//===================================================================//
// Ereigniskategorie - Alarmeldung - Meldung signalisiert Anlagenausfall oder erfordert sofortigen Eingriff 
// Event category - Alarm message - Message signals system failure or requires immediate intervention 
// Sicherheitstemperaturbegrenzer (STB), Sicherheitsdruckbegrenzer (SDB), Übertemperatur der Warmwasserbereitung (WWB), Sicherheitsventile, Hauptpumpen, Keilriemenwächter, Frequenzumformer, Kälteanlagen, Spannungsausfall usw
// Safety temperature limiter, safety pressure limiter, excess temperature of water heating, safety valves, main pumps, V-belt monitors, frequency converters, refrigeration systems, voltage failure, etc.
AlarmMsg.iParent							:= THIS^;
AlarmMsg.iLabel								:= LblControl_EvtCategoryAlarmMessage;									  
AlarmMsg.sObjectName						:= '{Idx=01}';
AlarmMsg.eDPADMode							:= E_BA_DPADMode.eInclude;																						
AlarmMsg.EC.nInstanceID							:= EC_ID.NC30;
AlarmMsg.EC.sObjectName							:= '{Idx=30}';
AlarmMsg.EC.eEventType							:= E_BA_EventType.eAlarm;
AlarmMsg.EC.aPriority[1]						:= 70;
AlarmMsg.EC.aPriority[2]						:= 71;
AlarmMsg.EC.aPriority[3]						:= 72;
AlarmMsg.EC.eAlarmMode						:= E_BA_AlarmMode.eExtended;	//Erweiterter Alarm


//===================================================================
// Ereigniskategorie - Störungsmeldung - Meldung weist auf einen anormalen Betriebszustand hin
// Event category - malfunction message - message indicates abnormal operating condition
// Temperaturwächter (TW), Druckwächter (DW), Temperaturüberwachung von Wärmetauscher (WT) und WWB, Motorschutz, Aufzug-Sammelstörmeldung, Netzdrücke usw.
// Temperature monitor, pressure monitor, temperature monitoring of heat exchanger and water heating, motor protection, lift collective fault signal, mains pressures, etc.
FaultMsg.iParent							:= THIS^;
FaultMsg.iLabel								:= LblControl_EvtCategoryFaultMessage;							  
FaultMsg.sObjectName						:= '{Idx=01}';
FaultMsg.eDPADMode							:= E_BA_DPADMode.eInclude;																						
FaultMsg.EC.nInstanceID							:= EC_ID.NC40;
FaultMsg.EC.sObjectName							:= '{Idx=40}';
FaultMsg.EC.eEventType							:= E_BA_EventType.eDisturb;
FaultMsg.EC.aPriority[1]						:= 100;
FaultMsg.EC.aPriority[2]						:= 101;
FaultMsg.EC.aPriority[3]						:= 102;
FaultMsg.EC.eAlarmMode						:= E_BA_AlarmMode.eStandard;	//Standard Alarm
//===================================================================
// Ereigniskategorie - Wartungsmeldung, Hinweis auf Wartungsaktivität o.ä.
// Event category - Maintenance message Maintenance message, indication of maintenance activity or similar.
// Betriebsstunden, Behälterstand, Reparaturschalter usw.
// Operating hours, tank level, repair switch, etc.
MaintenanceMsg01.iParent					:= THIS^;
MaintenanceMsg01.iLabel						:= LblControl_EvtCategoryMaintenanceMessage;									  
MaintenanceMsg01.sObjectName				:= '{Idx=01}';
MaintenanceMsg01.eDPADMode					:= E_BA_DPADMode.eInclude;																						
MaintenanceMsg01.EC.nInstanceID					:= EC_ID.NC50;
MaintenanceMsg01.EC.sObjectName					:= '{Idx=50}';
MaintenanceMsg01.EC.eEventType					:= E_BA_EventType.eMaintenance;
MaintenanceMsg01.EC.aPriority[1]				:= 130;
MaintenanceMsg01.EC.aPriority[2]				:= 131;
MaintenanceMsg01.EC.aPriority[3]				:= 132;
MaintenanceMsg01.EC.eAlarmMode						:= E_BA_AlarmMode.eStandard;	//Standard Alarm

// Filterende erreicht, Filter verschmutzt usw.
// Filter end reached, filter dirty, etc.
MaintenanceMsg02.iParent					:= THIS^;
MaintenanceMsg02.iLabel						:= LblControl_EvtCategoryMaintenanceMessage;									  
MaintenanceMsg02.sObjectName				:= '{Idx=02}';
MaintenanceMsg02.sDescription				:= '{Wartungsmeldung}';
MaintenanceMsg02.eDPADMode					:= E_BA_DPADMode.eInclude;																						
MaintenanceMsg02.EC.nInstanceID					:= EC_ID.NC51;
MaintenanceMsg02.EC.sObjectName					:= '{Idx=51}';
MaintenanceMsg02.EC.eEventType					:= E_BA_EventType.eAlarm;
MaintenanceMsg02.EC.aPriority[1]				:= 135;
MaintenanceMsg02.EC.aPriority[2]				:= 136;
MaintenanceMsg02.EC.aPriority[3]				:= 137;
MaintenanceMsg02.EC.eAlarmMode						:= E_BA_AlarmMode.eStandard;	//Standard Alarm
//===================================================================
//===================================================================
// Ereigniskategorie - Systemmeldung, Störungsmeldung aus GA-System
// Event category - System message, System message, Fault message from building automation system
// Gerätestörung, Batteriemeldung, Kommunikationsunterbrechung usw.
// Unit malfunction, battery message, communication interruption, etc.
SystemMsg.iParent							:= THIS^;
SystemMsg.iLabel							:= LblControl_EvtCategorySystem;									  
SystemMsg.sObjectName						:= '{Idx=01}';
SystemMsg.eDPADMode							:= E_BA_DPADMode.eInclude;																						
SystemMsg.EC.nInstanceID						:= EC_ID.NC60;
SystemMsg.EC.sObjectName						:= '{Idx=60}';
SystemMsg.EC.eEventType							:= E_BA_EventType.eNotification;
SystemMsg.EC.aPriority[1]						:= 180;
SystemMsg.EC.aPriority[2]						:= 181;
SystemMsg.EC.aPriority[3]						:= 182;
SystemMsg.EC.eAlarmMode						:= E_BA_AlarmMode.eSimple;	//Simple Alarm
//===================================================================//
//	Ereigniskategorie - Manual operation, Handeingriff
ManualOp.iParent							:= THIS^;
ManualOp.iLabel						 		:= LblControl_EvtCategoryManualOperation;									  
ManualOp.sObjectName						:= '{Idx=01}';
ManualOp.eDPADMode							:= E_BA_DPADMode.eInclude;																						
ManualOp.EC.nInstanceID							:= EC_ID.NC70;
ManualOp.EC.sObjectName							:= '{Idx=70}';
ManualOp.EC.eEventType							:= E_BA_EventType.eAlarm;
ManualOp.EC.aPriority[1]						:= 220;
ManualOp.EC.aPriority[2]						:= 220;
ManualOp.EC.aPriority[3]						:= 220;
ManualOp.EC.eAlarmMode						:= E_BA_AlarmMode.eSimple;	//Simple Alarm
//===================================================================//
// Ereigniskategorie - Freibleibend, Sonstige Meldungen
// Event category - Other message, Not binding, Other messages
// Betriebszustandswechsel, Betriebsarten, Trendspeicher voll usw.
// Operating status change, operating modes, trend memory full, etc.
OtherMsg.iParent							:= THIS^;
OtherMsg.iLabel						 		:= LblControl_EvtCategoryOther;									  
OtherMsg.sObjectName						:= '{Idx=01}';
OtherMsg.eDPADMode							:= E_BA_DPADMode.eInclude;																						
OtherMsg.EC.nInstanceID							:= EC_ID.NC80;
OtherMsg.EC.sObjectName							:= '{Idx=80}';
OtherMsg.EC.eEventType							:= E_BA_EventType.eAlarm;
OtherMsg.EC.aPriority[1]						:= 230;
OtherMsg.EC.aPriority[2]						:= 231;
OtherMsg.EC.aPriority[3]						:= 232;
OtherMsg.EC.eAlarmMode						:= E_BA_AlarmMode.eSimple;	//Simple Alarm
END_METHOD

END_FUNCTION_BLOCK

// ---- Templates/POUs/Universal/Control/EventClasses/FB_BA_EvtCategory.TcPOU
{region '#Template'}
	{attribute 'Version' := '1.2.1.0'}
	{attribute 'Tags' := '"LCID": "1031", "Text": "Universal, Control, Event class, Notification"'}
	{attribute 'Tags' := '"LCID": "1033", "Text": "Universal, Control, Event class, Notification"'}
	{attribute 'Using' := '"Type": "Template", "URI": "EC_AMEV"'}
	{attribute 'Description' := '"LCID": "1031", "Text": "Ereignisklasse"'}
	{attribute 'Description' := '"LCID": "1033", "Text": "Event class"'}
{endregion}
FUNCTION_BLOCK FB_BA_EvtCategory EXTENDS FB_BA_View
VAR_INPUT CONSTANT
		EC				: FB_BA_EC;  
END_VAR

SUPER^(); // FB_BA_View
EC(); // FB_BA_EC

METHOD FB_init : BOOL
VAR_INPUT
	bInitRetains : BOOL; // if TRUE, the retain variables are initialized (warm start / cold start)
	bInCopyCode : BOOL;  // if TRUE, the instance afterwards gets moved into the copy code (online change)
END_VAR
EC.iParent					:= THIS^;
EC.iLabel					:= LblControl_EvtClass;	
EC.nInstanceID				:= EC_ID.NC10;
EC.sObjectName				:= '{Idx=10}';
EC.eEventType				:= E_BA_EventType.eAlarm;
EC.aPriority[1]				:= 16;
EC.aPriority[2]				:= 17;
EC.aPriority[3]				:= 18;
END_METHOD

END_FUNCTION_BLOCK

// ---- Templates/POUs/Trade/General/Settings/FB_BA_Settings.TcPOU
{region '#Template'}
	{attribute 'Version' := '1.2.0.0'}
	{attribute 'Tags' := '"LCID": "1031", "Text": "General, Settings, Parameters, Basics"'}
	{attribute 'Tags' := '"LCID": "1033", "Text": "General, Settings, Parameters, Basics"'}
	{attribute 'Description' := '"LCID": "1031", "Text": "Basis Parameter für die Templates"'}
	{attribute 'Description' := '"LCID": "1033", "Text": "Basic parameters for the templates"'}
{endregion}
FUNCTION_BLOCK FB_BA_Settings EXTENDS FB_BA_View
VAR_INPUT
	fTWth					: REAL;	//	Weather temperature
END_VAR
VAR_INPUT CONSTANT
	WthParam			: FB_BA_WeatherParamter;
END_VAR
VAR

	GeneralSettings			: FB_BA_RawPublisher;									
	stSettings				: ST_BA_GeneralSettings;
END_VAR
VAR // added by the converter: edge detectors and wires of the graphical bodies
    _s1 : ST_BA_GeneralSettings;
END_VAR

SUPER^(); // FB_BA_View
WthParam(fTWth := fTWth); // FB_BA_WeatherParamter
// compose _s1 : ST_BA_GeneralSettings
_s1.fFrostProtectionSetpoint := WthParam.fSpFrstProtec;
_s1.fTWthLowLimit := WthParam.fTWthLowLimit;
_s1.bTWthLowLimit := WthParam.bTWthLowLimit;
_s1.fTWthDamped := WthParam.fTWthDamped;
_s1.bTWthDampedLowLimit := WthParam.bTWthDampedLowLimit;
_s1.fTWth := fTWth;
GeneralSettings(xData := _s1); // FB_BA_RawPublisher

METHOD FB_init : BOOL
VAR_INPUT
	bInitRetains : BOOL; // if TRUE, the retain variables are initialized (warm start / cold start)
	bInCopyCode : BOOL;  // if TRUE, the instance afterwards gets moved into the copy code (online change)
END_VAR
WthParam.iParent				:= THIS^;
WthParam.iLabel					:= LblCmpGeneral.Settings_WthParam;
WthParam.sObjectName			:= '{Idx=01}';
WthParam.eDPADMode				:= E_BA_DPADMode.eInclude;
END_METHOD

END_FUNCTION_BLOCK

// ---- Templates/POUs/Trade/General/Settings/FB_BA_WeatherParamter.TcPOU
{region '#Template'}
	{attribute 'Version' := '1.2.1.0'}
	{attribute 'Tags' := '"LCID": "1031", "Text": "General, Settings, Parameters, Basics"'}
	{attribute 'Tags' := '"LCID": "1033", "Text": "General, Settings, Parameters, Basics"'}
	{attribute 'Using' := '"Type": "Template", "URI": "BA2_Param"'}
	{attribute 'Description' := '"LCID": "1031", "Text": "Witterungsparameter für die Templates"'}
	{attribute 'Description' := '"LCID": "1033", "Text": "Weather parameters for the templates"'}
{endregion}
FUNCTION_BLOCK FB_BA_WeatherParamter EXTENDS FB_BA_View
VAR_INPUT
	fTWth					: REAL;	//	Weather temperature
END_VAR
VAR_OUTPUT
	fSpFrstProtec			: REAL;  // frost protection setpoint. for eg. Heating circutis in protection mode
	fTWthLowLimit			: REAL;  // below this value all frostprotection funcktions in HVAC-Plants will be enabled
	bTWthLowLimit			: BOOL;  // is TRUE when the outside temperature is below the value from fTWthLowLimit 
	fTWthDamped				: REAL;  // damped outside temperature
	bTWthDampedLowLimit		: BOOL;	
END_VAR
VAR_INPUT CONSTANT
	SpFrstProtec			: FB_BA_AV_Op;		
	TWthLowLimitVal			: FB_BA_AV_Op;																
	TWthLowLimit			: FB_BA_BV_Op;								
	TWthDamped				: FB_BA_AV_Op;		
	TWthDampedLowLimit		: FB_BA_BV_Op;	
END_VAR
VAR
	TWthLowLimitHys			: FB_BA_Swi2P;
	Average					: FB_BA_TiAvrg;
	DlyEn					: TON;
	TWthDampedLowLimitHys	: FB_BA_Swi2P;
END_VAR

SUPER^(); // FB_BA_View
SpFrstProtec(); // FB_BA_AV_Op
fSpFrstProtec := SpFrstProtec.fPresentValue;
TWthLowLimitVal(); // FB_BA_AV_Op
fTWthLowLimit := TWthLowLimitVal.fPresentValue;
TWthLowLimitHys(bEn := TRUE, fIn := fTWth, fOn := fTWthLowLimit, fOff := fTWthLowLimit + 1); // FB_BA_Swi2P
TWthLowLimit(bValuePgm := TWthLowLimitHys.bQ); // FB_BA_BV_Op
bTWthLowLimit := TWthLowLimit.bPresentValue;
DlyEn(IN := TRUE, PT := T#2s); // TON
Average(bEn := DlyEn.Q, fIn := fTWth, nIntval := 900, nNumOfElem := 96); // FB_BA_TiAvrg
TWthDamped(fValuePgm := Average.fOut); // FB_BA_AV_Op
fTWthDamped := TWthDamped.fPresentValue;
TWthDampedLowLimitHys(bEn := TRUE, fIn := fTWthDamped, fOn := fTWthLowLimit, fOff := fTWthLowLimit + 1.0); // FB_BA_Swi2P
TWthDampedLowLimit(bValuePgm := TWthDampedLowLimitHys.bQ); // FB_BA_BV_Op
bTWthDampedLowLimit := TWthDampedLowLimit.bPresentValue;

METHOD FB_init : BOOL
VAR_INPUT
	bInitRetains : BOOL; // if TRUE, the retain variables are initialized (warm start / cold start)
	bInCopyCode : BOOL;  // if TRUE, the instance afterwards gets moved into the copy code (online change)
END_VAR
SpFrstProtec.iParent				:= THIS^;
SpFrstProtec.iLabel					:= LblCmpGeneral.WthParam_SpFrstProtec;
SpFrstProtec.sObjectName			:= '{Idx=01}';
SpFrstProtec.eUnit					:= E_BA_Unit.eTemperature_DegreesCelsius;  
SpFrstProtec.fValueRm				:= 5.0;
SpFrstProtec.fCOVIncrement			:= BA2_Param.fDefCOVIncrement;							

TWthLowLimitVal.iParent				:= THIS^;
TWthLowLimitVal.iLabel				:= LblCmpGeneral.WthParam_TWthLowLimitVal;
TWthLowLimitVal.sObjectName			:= '{Idx=01}';
TWthLowLimitVal.eUnit				:= E_BA_Unit.eTemperature_DegreesCelsius;  
TWthLowLimitVal.fValueRm			:= 8.0;
TWthLowLimitVal.fCOVIncrement		:= BA2_Param.fDefCOVIncrement;							

TWthLowLimit.iParent				:= THIS^;		
TWthLowLimit.iLabel 				:= LblCmpGeneral.WthParam_TWthLowLimit;	
TWthLowLimit.sObjectName			:= '{Idx=01}';												
TWthLowLimit.sInactiveText			:= txtEvent_Off;
TWthLowLimit.sActiveText			:= txtEvent_On;
TWthLowLimit.bValueRm				:= FALSE;		
TWthLowLimit.eToggleMode 			:= E_BA_ToggleMode.eSwitch;

TWthDamped.iParent					:= THIS^;
TWthDamped.iLabel					:= LblCmpGeneral.WthParam_TWthDamped;
TWthDamped.sObjectName				:= '{Idx=01}';
TWthDamped.eUnit					:= E_BA_Unit.eTemperature_DegreesCelsius;  
TWthDamped.fValueRm					:= 0.0;
TWthDamped.fCOVIncrement			:= BA2_Param.fDefCOVIncrement;							


TWthDampedLowLimit.iParent			:= THIS^;		
TWthDampedLowLimit.iLabel 			:= LblCmpGeneral.WthParam_TWthDampedLowLimit;	
TWthDampedLowLimit.sObjectName		:= '{Idx=02}';												
TWthDampedLowLimit.sInactiveText	:= txtEvent_Off;
TWthDampedLowLimit.sActiveText		:= txtEvent_On;
TWthDampedLowLimit.bValueRm			:= FALSE;								
TWthDampedLowLimit.eToggleMode 		:= E_BA_ToggleMode.eSwitch;
END_METHOD

END_FUNCTION_BLOCK

// ---- Templates/POUs/Trade/General/ControlCabinet/FB_BA_ControlCabinet.TcPOU
{region '#Template'}
	{attribute 'Version' := '1.2.1.0'}
	{attribute 'Tags' := '"LCID": "1031", "Text": "General, Cabinet, Control cabinet"'}
	{attribute 'Tags' := '"LCID": "1033", "Text": "General, Cabinet, Control cabinet"'}
	{attribute 'Using' := '"Type": "Template", "URI": "EC_AMEV"'}
	{attribute 'Description' := '"LCID": "1031", "Text": "Schaltschrank Ereignisse"'}
	{attribute 'Description' := '"LCID": "1033", "Text": "Control cabinet events"'}
{endregion}
FUNCTION_BLOCK FB_BA_ControlCabinet EXTENDS FB_BA_ControlCabinetBasic
VAR_INPUT CONSTANT
	Fuse01					: FB_BA_SensorBinary_IO;		
	Fuse02					: FB_BA_SensorBinary_IO;	
	Fuse03					: FB_BA_SensorBinary_IO;	
END_VAR

SUPER^(); // FB_BA_ControlCabinetBasic
Fuse01(); // FB_BA_SensorBinary_IO
Fuse02(); // FB_BA_SensorBinary_IO
Fuse03(); // FB_BA_SensorBinary_IO

METHOD FB_init : BOOL
VAR_INPUT
	bInitRetains : BOOL; // if TRUE, the retain variables are initialized (warm start / cold start)
	bInCopyCode : BOOL;  // if TRUE, the instance afterwards gets moved into the copy code (online change)
END_VAR
Fuse01.iParent								:= THIS^;		
Fuse01.iLabel 								:= LblCmpGeneral.ControlCabinet_Fuse;	
Fuse01.sObjectName							:= '{Idx=01}';
Fuse01.eDPADMode							:= E_BA_DPADMode.eInclude;																						
Fuse01.Input.iLabel							:= LblCmpGeneral.ControlCabinet_Fuse_Input;	
Fuse01.Input.sObjectName					:= '{Idx=01}';	
Fuse01.Input.ePolarity						:= E_BA_Polarity.eReverse;
Fuse01.Input.sActiveText 					:= txtEvent_Triggered;
Fuse01.Input.sInactiveText 					:= txtEvent_Normal;
Fuse01.Input.nEventClassID					:= EC_ID.NC30;
Fuse01.Input.aEventTransitionText[1]		:= txtEvent_Triggered;
Fuse01.Input.aEventTransitionText[2]		:= txtEvent_Error;
Fuse01.Input.aEventTransitionText[3]		:= txtEvent_Normal;
Fuse01.Input.bEventDetectionEnable			:= TRUE;
Fuse01.Input.aEventEnable[1]				:= TRUE;			//	to_offnormal
Fuse01.Input.aEventEnable[2]				:= TRUE;			//	to_fault
Fuse01.Input.aEventEnable[3]				:= TRUE;			//	to_normal
Fuse01.Input.eEnPlantLock					:= E_BA_LockPriority.eNoLock;	
								 
Fuse02.iParent								:= THIS^;		
Fuse02.iLabel 								:= LblCmpGeneral.ControlCabinet_Fuse;	
Fuse02.sObjectName							:= '{Idx=02}';
Fuse02.eDPADMode							:= E_BA_DPADMode.eInclude;																						
Fuse02.Input.iLabel							:= LblCmpGeneral.ControlCabinet_Fuse_Input;	
Fuse02.Input.sObjectName					:= '{Idx=02}';	
Fuse02.Input.ePolarity						:= E_BA_Polarity.eReverse;
Fuse02.Input.sActiveText 					:= txtEvent_Triggered;
Fuse02.Input.sInactiveText 					:= txtEvent_Normal;
Fuse02.Input.nEventClassID					:= EC_ID.NC30;
Fuse02.Input.aEventTransitionText[2]		:= txtEvent_Error;
Fuse02.Input.aEventTransitionText[3]		:= txtEvent_Normal;
Fuse02.Input.bEventDetectionEnable			:= TRUE;
Fuse02.Input.aEventEnable[1]				:= TRUE;			//	to_offnormal
Fuse02.Input.aEventEnable[2]				:= TRUE;			//	to_fault
Fuse02.Input.aEventEnable[3]				:= TRUE;			//	to_normal
Fuse02.Input.eEnPlantLock					:= E_BA_LockPriority.eNoLock;	
										 
Fuse03.iParent								:= THIS^;		
Fuse03.iLabel 								:= LblCmpGeneral.ControlCabinet_Fuse;	
Fuse03.sObjectName							:= '{Idx=03}';
Fuse03.eDPADMode							:= E_BA_DPADMode.eInclude;																						
Fuse03.Input.iLabel							:= LblCmpGeneral.ControlCabinet_Fuse_Input;	
Fuse03.Input.sObjectName					:= '{Idx=03}';	
Fuse03.Input.ePolarity						:= E_BA_Polarity.eReverse;
Fuse03.Input.sActiveText 					:= txtEvent_Triggered;
Fuse03.Input.sInactiveText 					:= txtEvent_Normal;
Fuse03.Input.nEventClassID					:= EC_ID.NC30;
Fuse03.Input.aEventTransitionText[1]		:= txtEvent_Triggered;
Fuse03.Input.aEventTransitionText[2]		:= txtEvent_Error;
Fuse03.Input.aEventTransitionText[3]		:= txtEvent_Normal;
Fuse03.Input.bEventDetectionEnable			:= TRUE;
Fuse03.Input.aEventEnable[1]				:= TRUE;			//	to_offnormal
Fuse03.Input.aEventEnable[2]				:= TRUE;			//	to_fault
Fuse03.Input.aEventEnable[3]				:= TRUE;			//	to_normal
Fuse03.Input.eEnPlantLock					:= E_BA_LockPriority.eNoLock;
END_METHOD

END_FUNCTION_BLOCK

// ---- Templates/POUs/Trade/General/ControlCabinet/FB_BA_ControlCabinetBasic.TcPOU
{region '#Template'}
	{attribute 'Version' := '1.2.1.0'}
	{attribute 'Tags' := '"LCID": "1031", "Text": "General, Cabinet, Control cabinet, Acknowledgement"'}
	{attribute 'Tags' := '"LCID": "1033", "Text": "General, Cabinet, Control cabinet, Acknowledgement"'}
	{attribute 'Using' := '"Type": "Template", "URI": "EC_AMEV"'}
	{attribute 'Description' := '"LCID": "1031", "Text": "Schaltschrank Quittierung"'}
	{attribute 'Description' := '"LCID": "1033", "Text": "Control cabinet acknowledgement"'}
{endregion}
FUNCTION_BLOCK FB_BA_ControlCabinetBasic EXTENDS FB_BA_View
VAR
	// By default, the entire project structure can be acknowledged.
	// There may be constellations (e.g. multiple control cabinets) where only one part of the project structure (e.g. multiple buildings) has to be acknowledged.
	// > In this case separete parts can be assigned here: 
	iAckView1				: I_BA_View;
	iAckView2				: I_BA_View;
	iAckView3				: I_BA_View;
END_VAR
VAR_INPUT CONSTANT
	LampFault				: FB_BA_ActuatorCmd;		
	AckButton				: FB_BA_CombinationBI_BV;													
	RstHw					: FB_BA_ActuatorCmd;														
END_VAR
VAR				
	bIsDisturbed			: BOOL;
	bHasUnackEvent			: BOOL;
	bBlink					: BOOL;
	tAlmLampImpuls			: FB_BA_Blink;						
	tpResetHw				: TP;	
	rtrigRstSwi				: R_TRIG;
	bTrigRstSwi				: BOOL;
	rtrigRstButton			: R_TRIG;
	bTrigRstButton			: BOOL;	
END_VAR

SUPER^(); // FB_BA_View
EventEvaluation();
LampFault(bEnPgm := bIsDisturbed, bValPgm := SEL(bHasUnackEvent, TRUE, bBlink)); // FB_BA_ActuatorCmd
AckButton(); // FB_BA_CombinationBI_BV
rtrigRstSwi(CLK := AckButton.bBI_PrVal); // R_TRIG
bTrigRstSwi := rtrigRstSwi.Q;
rtrigRstButton(CLK := AckButton.bBV_PrVal); // R_TRIG
bTrigRstButton := rtrigRstButton.Q;
tpResetHw(IN := bTrigRstSwi OR bTrigRstButton, PT := T#2s); // TP
RstHw(bEnPgm := TRUE, bValPgm := tpResetHw.Q); // FB_BA_ActuatorCmd

METHOD PRIVATE Ack
VAR_INPUT
	iView			: I_BA_View;
END_VAR
IF (iView <> 0) THEN
	iView.AcknowledgeObjectsPLC := (bTrigRstSwi) OR (bTrigRstButton);	
END_IF
END_METHOD

METHOD PRIVATE EventEvaluation
VAR
	_iView			: I_BA_View;
END_VAR
bIsDisturbed := FALSE;
bHasUnackEvent := FALSE;

IF (iAckView1 = 0) AND (iAckView2 = 0) AND (iAckView3 = 0) THEN
	// Treat project structure via root-object:
	Ack(XBA_Globals.Top);
	GetErrors(XBA_Globals.Top);
ELSE
	// Treat each defined object:
	Ack(iAckView1);
	GetErrors(iAckView1);
	
	Ack(iAckView2);
	GetErrors(iAckView2);
	
	Ack(iAckView3);
	GetErrors(iAckView3);
END_IF

// Generate alarm lamp impulse:
tAlmLampImpuls();

bBlink := tAlmLampImpuls.bQ;
END_METHOD

METHOD FB_init : BOOL
VAR_INPUT
	bInitRetains : BOOL; // if TRUE, the retain variables are initialized (warm start / cold start)
	bInCopyCode : BOOL;  // if TRUE, the instance afterwards gets moved into the copy code (online change)
END_VAR
LampFault.iParent							:= THIS^;
LampFault.iLabel							:= LblCmpGeneral.ControlCabinet_LampFault;			
LampFault.sObjectName						:= '{Idx=01}';
LampFault.eDPADMode							:= E_BA_DPADMode.eInclude;																						
LampFault.Cmd.iLabel						:= LblCmpGeneral.ControlCabinet_LampFault_Cmd;			
LampFault.Cmd.sObjectName					:= '{Idx=01}';	
LampFault.Cmd.ePolarity						:= E_BA_Polarity.eNormal;
LampFault.Cmd.eFeedbackPolarity				:= E_BA_Polarity.eNormal;
LampFault.Cmd.eOverriddenPolarity			:= E_BA_Polarity.eReverse;
LampFault.Cmd.sActiveText 					:= txtEvent_On;
LampFault.Cmd.sInactiveText 				:= txtEvent_Off;
LampFault.Cmd.nEventClassID					:= EC_ID.NC40;
LampFault.Cmd.aEventTransitionText[1]		:= txtEvent_Disturb;
LampFault.Cmd.aEventTransitionText[2]		:= txtEvent_None;
LampFault.Cmd.aEventTransitionText[3]		:= txtEvent_Normal;
LampFault.Cmd.bEventDetectionEnable			:= FALSE;
LampFault.Cmd.eEnPlantLock					:= E_BA_LockPriority.eNoLock;	

AckButton.iParent							:= THIS^;		
AckButton.iLabel 							:= LblCmpGeneral.ControlCabinet_AckButton;	
AckButton.sObjectName						:= '{Idx=01}';
AckButton.eDPADMode							:= E_BA_DPADMode.eInclude;																						
AckButton.Input.iLabel						:= LblCmpGeneral.ControlCabinet_AckButton_Input;
AckButton.Input.ePolarity					:= E_BA_Polarity.eNormal;
AckButton.Input.bEventDetectionEnable		:= FALSE;
AckButton.Value.iLabel						:= LblCmpGeneral.ControlCabinet_AckButton_Value;
AckButton.Value.eToggleMode 				:= E_BA_ToggleMode.ePushButton;									

RstHw.iParent								:= THIS^;
RstHw.iLabel								:= LblCmpGeneral.ControlCabinet_RstHw;			
RstHw.sObjectName							:= '{Idx=02}';
RstHw.eDPADMode								:= E_BA_DPADMode.eInclude;																						
RstHw.Cmd.iLabel							:= LblCmpGeneral.ControlCabinet_RstHw_Cmd;			
RstHw.Cmd.sObjectName						:= '{Idx=01}';	
RstHw.Cmd.ePolarity							:= E_BA_Polarity.eNormal;
RstHw.Cmd.eFeedbackPolarity					:= E_BA_Polarity.eNormal;
RstHw.Cmd.eOverriddenPolarity				:= E_BA_Polarity.eReverse;
RstHw.Cmd.sActiveText 						:= txtEvent_On;
RstHw.Cmd.sInactiveText 					:= txtEvent_Off;
RstHw.Cmd.nEventClassID						:= EC_ID.NC40;
RstHw.Cmd.aEventTransitionText[1]			:= txtEvent_Disturb;
RstHw.Cmd.aEventTransitionText[2]			:= txtEvent_None;
RstHw.Cmd.aEventTransitionText[3]			:= txtEvent_Normal;
RstHw.Cmd.bEventDetectionEnable				:= FALSE;
RstHw.Cmd.eEnPlantLock						:= E_BA_LockPriority.eNoLock;	

tAlmLampImpuls.bEn							:=	TRUE; 
tAlmLampImpuls.nTiOn						:=	800;
tAlmLampImpuls.nTiOff						:=	800;
END_METHOD

METHOD PRIVATE GetErrors
VAR_INPUT
	iView			: I_BA_View;
END_VAR
VAR
	iTemp			: INT;
	fbEvents		: REFERENCE TO FB_BA_EventIndicator;
END_VAR
IF (iView <> 0) THEN
	fbEvents REF= iView.ActiveEvents;
	
	FOR iTemp := E_BA_EventType.First TO E_BA_EventType.Last DO
		IF (fbEvents.aEventsPerIconImage[iTemp].nCount > 0) THEN
			bIsDisturbed := TRUE;
			
			CASE (fbEvents.aEventsPerIconImage[iTemp].eMostPriorisedState) OF
				E_BA_EventIconState.ePresent,
				E_BA_EventIconState.eGone:
					bHasUnackEvent := TRUE;
			END_CASE
		END_IF
	END_FOR
END_IF
END_METHOD

METHOD PROTECTED Reset
VAR_INPUT
	bUnregister			: BOOL			:= FALSE;
END_VAR
iAckView1 := 0;
iAckView2 := 0;
iAckView3 := 0;

SUPER^.Reset(bUnregister);
END_METHOD

END_FUNCTION_BLOCK

// ---- Templates/POUs/Universal/Aggregat/Binary/FB_BA_ActuatorCmd.TcPOU
{region '#Template'}
	{attribute 'Version' := '1.2.1.0'}
	{attribute 'Tags' := '"LCID": "1031", "Text": "Universal, Analog, Aggregate"'}
	{attribute 'Tags' := '"LCID": "1033", "Text": "Universal, Analog, Aggregate"'}
	{attribute 'Using' := '"Type": "Template", "URI": "EC_AMEV"'}
	{attribute 'Using' := '"Type": "Template", "URI": "BA2_Param"'}
	{attribute 'Description' := '"LCID": "1031", "Text": "Aktor binär"'}
	{attribute 'Description' := '"LCID": "1033", "Text": "Actuator binary"'}
{endregion}
FUNCTION_BLOCK FB_BA_ActuatorCmd EXTENDS FB_BA_AggregateB
VAR_OUTPUT
	bCmd							: BOOL;
END_VAR
VAR_INPUT CONSTANT
	Cmd						: FB_BA_BO_IO;			
END_VAR

SUPER^(); // FB_BA_AggregateB
Cmd(
    bEnSfty := bEnSfty,
    bValSfty := SUPER^.bActiveVal,
    bEnCrit := bEnCrit,
    bValCrit := SUPER^.bActiveVal,
    bEnPgm := bEnPgm,
    bValPgm := SUPER^.bActiveVal); // FB_BA_BO_IO
bCmd := Cmd.bPresentValue;

METHOD FB_init : BOOL
VAR_INPUT
	bInitRetains : BOOL; // if TRUE, the retain variables are initialized (warm start / cold start)
	bInCopyCode : BOOL;  // if TRUE, the instance afterwards gets moved into the copy code (online change)
END_VAR
Cmd.iParent							:= THIS^;
Cmd.iLabel							:= LblUniFieldDevice.Aggregat_Cmd;			
Cmd.sObjectName						:= '{Idx=01}';	
Cmd.sDeviceType						:= '';
Cmd.bEnOutOfService					:= FALSE;
Cmd.ePolarity						:= E_BA_Polarity.eNormal;
Cmd.eFeedbackPolarity				:= E_BA_Polarity.eNormal;
Cmd.eOverriddenPolarity				:= E_BA_Polarity.eReverse;
Cmd.sActiveText 					:= txtEvent_On;
Cmd.sInactiveText 					:= txtEvent_Off;
Cmd.nStateChangeCount				:= 0;
Cmd.nActiveTimeElapsed				:= 0;
Cmd.nMinimumOnTime					:= 0;
Cmd.nMinimumOffTime					:= 0;
Cmd.bEnManualRm						:= FALSE;	//	Priority  8	
Cmd.bValManualRm					:= FALSE;	//	Priority  8
Cmd.bDefaultValue					:= FALSE;
Cmd.nEventClassID					:= EC_ID.NC40;
Cmd.stTimeDelay.nToNormal			:= BA2_Param.nDefTimeDelay_ToNormal;
Cmd.stTimeDelay.nToAbnormal			:= BA2_Param.nDefTimeDelay_ToAbnormal;
Cmd.bAcknowledgeRm					:= FALSE;		
Cmd.aEventTransitionText[1]			:= txtEvent_Disturb;
Cmd.aEventTransitionText[2]			:= txtEvent_None;
Cmd.aEventTransitionText[3]			:= txtEvent_Normal;
Cmd.bEventDetectionEnable			:= FALSE;
Cmd.aEventEnable[1]					:= TRUE;			//	to_offnormal
Cmd.aEventEnable[2]					:= TRUE;			//	to_fault
Cmd.aEventEnable[3]					:= TRUE;			//	to_normal
Cmd.eEnPlantLock					:= E_BA_LockPriority.eNoLock;
END_METHOD

END_FUNCTION_BLOCK

// ---- Templates/POUs/Universal/Sensor/FB_BA_CombinationBI_BV.TcPOU
{region '#Template'}
	{attribute 'Version' := '1.2.1.0'}
	{attribute 'Tags' := '"LCID": "1031", "Text": "Universal, Sensor, BI, BV"'}
	{attribute 'Tags' := '"LCID": "1033", "Text": "Universal, Sensor, BI, BV"'}
	{attribute 'Using' := '"Type": "Template", "URI": "EC_AMEV"'}
	{attribute 'Using' := '"Type": "Template", "URI": "BA2_Param"'}
	{attribute 'Description' := '"LCID": "1031", "Text": "Kombination aus BV BI"'}
	{attribute 'Description' := '"LCID": "1033", "Text": "Combination of BV BI"'}
{endregion}	 
FUNCTION_BLOCK FB_BA_CombinationBI_BV EXTENDS FB_BA_View
VAR_INPUT
END_VAR
VAR_INPUT CONSTANT
	Input				: FB_BA_BI_IO;	
	Value				: FB_BA_BV_Op;									
END_VAR
VAR_OUTPUT
	bBI_PrVal			: BOOL;
	bBV_PrVal			: BOOL;	
END_VAR
VAR
END_VAR

SUPER^(); // FB_BA_View
Input(); // FB_BA_BI_IO
bBI_PrVal := Input.bPresentValue;
Value(); // FB_BA_BV_Op
bBV_PrVal := Value.bPresentValue;

METHOD FB_init : BOOL
VAR_INPUT
	bInitRetains : BOOL; // if TRUE, the retain variables are initialized (warm start / cold start)
	bInCopyCode : BOOL;  // if TRUE, the instance afterwards gets moved into the copy code (online change)
END_VAR
Input.iParent						:= THIS^;
Input.iLabel						:= LblFunctions_Button;	
Input.sObjectName					:= '{Idx=01}';
Input.sDeviceType					:= '';	
Input.bEnOutOfService				:= FALSE;
Input.ePolarity						:= E_BA_Polarity.eReverse;
Input.sActiveText 					:= txtEvent_On;
Input.sInactiveText 				:= txtEvent_Off;
Input.nStateChangeCount				:= 0;
Input.nActiveTimeElapsed			:= 0;
Input.nEventClassID					:= EC_ID.NC80;
Input.stTimeDelay.nToNormal			:= BA2_Param.nDefTimeDelay_ToNormal;
Input.stTimeDelay.nToAbnormal		:= BA2_Param.nDefTimeDelay_ToAbnormal;
Input.bAlarmValue					:= TRUE;
Input.bAcknowledgeRm				:= FALSE;		
Input.aEventTransitionText[1]		:= txtEvent_Off;
Input.aEventTransitionText[2]		:= txtEvent_None;
Input.aEventTransitionText[3]		:= txtEvent_On;
Input.bEventDetectionEnable			:= FALSE;
Input.aEventEnable[1]				:= TRUE;			//	to_offnormal
Input.aEventEnable[2]				:= TRUE;			//	to_fault
Input.aEventEnable[3]				:= TRUE;			//	to_normal
Input.eEnPlantLock					:= E_BA_LockPriority.eNoLock;	

Value.iParent						:= THIS^;		
Value.iLabel 						:= LblFunctions_Button;	
Value.sObjectName					:= '{Idx=02}';	
Value.sActiveText					:= txtEvent_On;
Value.sInactiveText					:= txtEvent_Off;
Value.bValueRm						:= FALSE;
Value.eToggleMode 					:= E_BA_ToggleMode.eSwitch;
END_METHOD

END_FUNCTION_BLOCK

// ---- Templates/POUs/Universal/Sensor/FB_BA_SensorBinary_IO.TcPOU
{region '#Template'}
	{attribute 'Version' := '1.2.1.0'}
	{attribute 'Tags' := '"LCID": "1031", "Text": "Universal, Sensor, BI"'}
	{attribute 'Tags' := '"LCID": "1033", "Text": "Universal, Sensor, BI"'}
	{attribute 'Using' := '"Type": "Template", "URI": "EC_AMEV"'}
	{attribute 'Using' := '"Type": "Template", "URI": "BA2_Param"'}
	{attribute 'Description' := '"LCID": "1031", "Text": "BI mit IO"'}
	{attribute 'Description' := '"LCID": "1033", "Text": "BI with IO"'}
{endregion}		 
FUNCTION_BLOCK FB_BA_SensorBinary_IO EXTENDS FB_BA_View
VAR_INPUT
END_VAR
VAR_INPUT CONSTANT
	Input					: FB_BA_BI_IO;		
END_VAR
VAR_OUTPUT
	bPresentValue			: BOOL;	
END_VAR
VAR
END_VAR

SUPER^(); // FB_BA_View
Input(); // FB_BA_BI_IO
bPresentValue := Input.bPresentValue;

METHOD FB_init : BOOL
VAR_INPUT
	bInitRetains : BOOL; // if TRUE, the retain variables are initialized (warm start / cold start)
	bInCopyCode : BOOL;  // if TRUE, the instance afterwards gets moved into the copy code (online change)
END_VAR
Input.iParent						:= THIS^;
Input.iLabel						:= LblUniFieldDevice.SensorBinary_Input;	
Input.sObjectName					:= '{Idx=01}';	
Input.sDeviceType					:= '';
Input.bEnOutOfService				:= FALSE;
Input.ePolarity						:= E_BA_Polarity.eReverse;
Input.sActiveText 					:= txtEvent_Triggered;
Input.sInactiveText 				:= txtEvent_Normal;
Input.nStateChangeCount				:= 0;
Input.nActiveTimeElapsed			:= 0;
Input.nEventClassID					:= EC_ID.NC30;
Input.stTimeDelay.nToNormal			:= BA2_Param.nDefTimeDelay_ToNormal;
Input.stTimeDelay.nToAbnormal		:= BA2_Param.nDefTimeDelay_ToAbnormal;
Input.bAlarmValue					:= TRUE;
Input.bAcknowledgeRm				:= FALSE;		
Input.aEventTransitionText[1]		:= txtEvent_Triggered;
Input.aEventTransitionText[2]		:= txtEvent_Error;
Input.aEventTransitionText[3]		:= txtEvent_Normal;
Input.bEventDetectionEnable			:= TRUE;
Input.aEventEnable[1]				:= TRUE;			//	to_offnormal
Input.aEventEnable[2]				:= TRUE;			//	to_fault
Input.aEventEnable[3]				:= TRUE;			//	to_normal
Input.eEnPlantLock					:= E_BA_LockPriority.eNoLock;
END_METHOD

END_FUNCTION_BLOCK

// ---- Templates/POUs/Trade/General/Building/FB_BA_BuildingGlobal.TcPOU
{region '#Template'}
	{attribute 'Version' := '1.2.0.0'}
	{attribute 'Tags' := '"LCID": "1031", "Text": "General, Building"'}
	{attribute 'Tags' := '"LCID": "1033", "Text": "General, Building"'}
	{attribute 'Description' := '"LCID": "1031", "Text": "Aufruf Gebäude Funktionen"'}
	{attribute 'Description' := '"LCID": "1033", "Text": "Call building functions"'}
{endregion}
FUNCTION_BLOCK FB_BA_BuildingGlobal EXTENDS FB_BA_View
VAR_INPUT CONSTANT
	BuildAlm			: FB_BA_BuildingAlarms;
	BuildMode			: FB_BA_BuildingMode;
END_VAR

SUPER^(); // FB_BA_View
BuildAlm(); // FB_BA_BuildingAlarms
BuildMode(); // FB_BA_BuildingMode

METHOD FB_init : BOOL
VAR_INPUT
	bInitRetains : BOOL; // if TRUE, the retain variables are initialized (warm start / cold start)
	bInCopyCode : BOOL;  // if TRUE, the instance afterwards gets moved into the copy code (online change)
END_VAR
BuildAlm.iParent			:= THIS^;	
BuildAlm.iLabel				:= LblCmpGeneral.BuildingGlobal_BuildAlm;
BuildAlm.sObjectName		:= '{Idx=01}';											 
BuildAlm.eDPADMode			:= E_BA_DPADMode.eInclude;
                        
BuildMode.iParent			:= THIS^;	
BuildMode.iLabel			:= LblCmpGeneral.BuildingGlobal_BuildMode;
BuildMode.sObjectName		:= '{Idx=02}';											 
BuildMode.eDPADMode			:= E_BA_DPADMode.eInclude;
END_METHOD

END_FUNCTION_BLOCK

// ---- Templates/POUs/Trade/General/Building/FB_BA_BuildingAlarms.TcPOU
{region '#Template'}
	{attribute 'Version' := '1.2.1.0'}
	{attribute 'Tags' := '"LCID": "1031", "Text": "General, Alarms"'}
	{attribute 'Tags' := '"LCID": "1033", "Text": "General, Alarms"'}
	{attribute 'Using' := '"Type": "Template", "URI": "BA2_Param"'}
	{attribute 'Using' := '"Type": "Template", "URI": "EC_AMEV"'}
	{attribute 'Using' := '"Type": "Template", "URI": "ST_BA_BuildingAlarms"'}
	{attribute 'Description' := '"LCID": "1031", "Text": "Gebäude Alarme"'}
	{attribute 'Description' := '"LCID": "1031", "Text": "Gebäude Alarme"'}
	{attribute 'Description' := '"LCID": "1033", "Text": "Building alarms"'}
{endregion}
FUNCTION_BLOCK FB_BA_BuildingAlarms EXTENDS FB_BA_View
VAR_INPUT CONSTANT
	FireAlert			: FB_BA_BI_IO;                      
	Bgly				: FB_BA_BI_IO;
	CentSwiOff			: FB_BA_BV_Op;
END_VAR	
VAR		
	BuildingAlarms		: FB_BA_RawPublisher;
END_VAR
VAR // added by the converter: edge detectors and wires of the graphical bodies
    _s1 : ST_BA_BuildingAlarms;
END_VAR

SUPER^(); // FB_BA_View
FireAlert(); // FB_BA_BI_IO
Bgly(); // FB_BA_BI_IO
CentSwiOff(); // FB_BA_Bv_OP
// compose _s1 : ST_BA_BuildingAlarms
_s1.bBurglary := Bgly.bPresentValue;
_s1.bFireAlert := FireAlert.bPresentValue;
_s1.bCentralOff := CentSwiOff.bPresentValue;
_s1.bForcedVentilation := FALSE;
_s1.bSmokeExtraction := FALSE;
BuildingAlarms(xData := _s1); // FB_BA_RawPublisher

METHOD FB_init : BOOL
VAR_INPUT
	bInitRetains : BOOL; // if TRUE, the retain variables are initialized (warm start / cold start)
	bInCopyCode : BOOL;  // if TRUE, the instance afterwards gets moved into the copy code (online change)
END_VAR
FireAlert.iParent						:= THIS^;
FireAlert.iLabel						:= LblCmpGeneral.BuildingAlarms_FireAlert;	
FireAlert.sObjectName					:= '{Idx=01}';	
FireAlert.sDeviceType					:= '';
FireAlert.bEnOutOfService				:= FALSE;
FireAlert.ePolarity						:= E_BA_Polarity.eReverse;
FireAlert.sActiveText 					:= txtEvent_On;
FireAlert.sInactiveText 				:= txtEvent_Alert;
FireAlert.nStateChangeCount				:= 0;
FireAlert.nActiveTimeElapsed			:= 0;
FireAlert.nEventClassID					:= EC_ID.NC10;
FireAlert.stTimeDelay.nToNormal			:= BA2_Param.nDefTimeDelay_ToNormal;
FireAlert.stTimeDelay.nToAbnormal		:= BA2_Param.nDefTimeDelay_ToAbnormal;
FireAlert.bAlarmValue					:= TRUE;
FireAlert.bAcknowledgeRm				:= FALSE;	
FireAlert.aEventTransitionText[1]		:= txtEvent_Alert;
FireAlert.aEventTransitionText[2]		:= txtEvent_None;
FireAlert.aEventTransitionText[3]		:= txtEvent_Normal;
FireAlert.bEventDetectionEnable			:= TRUE;
FireAlert.aEventEnable[1]				:= TRUE;			//	to_offnormal
FireAlert.aEventEnable[2]				:= TRUE;			//	to_fault
FireAlert.aEventEnable[3]				:= TRUE;			//	to_normal
FireAlert.eEnPlantLock					:= E_BA_LockPriority.eNoLock;	

Bgly.iParent							:= THIS^;
Bgly.iLabel								:= LblCmpGeneral.BuildingAlarms_Bgly;	
Bgly.sObjectName						:= '{Idx=02}';	
Bgly.sDeviceType						:= '';
Bgly.bEnOutOfService					:= FALSE;
Bgly.ePolarity							:= E_BA_Polarity.eReverse;
Bgly.sActiveText 						:= txtEvent_On;
Bgly.sInactiveText 						:= txtEvent_Alert;
Bgly.nStateChangeCount					:= 0;
Bgly.nActiveTimeElapsed					:= 0;
Bgly.nEventClassID						:= EC_ID.NC10;
Bgly.stTimeDelay.nToNormal				:= BA2_Param.nDefTimeDelay_ToNormal;
Bgly.stTimeDelay.nToAbnormal			:= BA2_Param.nDefTimeDelay_ToAbnormal;
Bgly.bAlarmValue						:= TRUE;
Bgly.bAcknowledgeRm						:= FALSE;	
Bgly.aEventTransitionText[1]			:= txtEvent_Alert;
Bgly.aEventTransitionText[2]			:= txtEvent_None;
Bgly.aEventTransitionText[3]			:= txtEvent_Normal; 
Bgly.bEventDetectionEnable				:= TRUE;
Bgly.aEventEnable[1]					:= TRUE;			//	to_offnormal
Bgly.aEventEnable[2]					:= TRUE;			//	to_fault
Bgly.aEventEnable[3]					:= TRUE;			//	to_normal
Bgly.eEnPlantLock						:= E_BA_LockPriority.eNoLock;	
                       	
CentSwiOff.iParent						:= THIS^;
CentSwiOff.iLabel 						:= LblCmpGeneral.BuildingAlarms_CentSwiOff;	
CentSwiOff.sObjectName					:= '{Idx=01}';
CentSwiOff.sInactiveText				:= txtEvent_Off;
CentSwiOff.sActiveText					:= txtEvent_On;
CentSwiOff.bValueRm						:= FALSE;
CentSwiOff.eToggleMode					:= E_BA_ToggleMode.ePushButton;
END_METHOD

END_FUNCTION_BLOCK

// ---- Templates/POUs/Trade/General/Building/FB_BA_BuildingMode.TcPOU
{region '#Template'}
	{attribute 'Version' := '1.2.1.0'}
	{attribute 'Tags' := '"LCID": "1031", "Text": "General, Building, Operating mode"'}
	{attribute 'Tags' := '"LCID": "1033", "Text": "General, Building, Operating mode"'}
	{attribute 'Description' := '"LCID": "1031", "Text": "Gebäude Betriebsart"'}
	{attribute 'Description' := '"LCID": "1033", "Text": "Building operating mode"'}
{endregion}
FUNCTION_BLOCK FB_BA_BuildingMode EXTENDS FB_BA_View
VAR_INPUT CONSTANT
	OpModMan					: FB_BA_MV_Op;
	OpModPr						: FB_BA_MV_Op;
	Sched						: FB_BA_SchedM;
END_VAR
VAR	
	DeMuxManMod					: FB_BA_DMUX_B04;		
	DeMuxSched					: FB_BA_DMUX_B04;		
	PrioSwi						: FB_BA_PrioSwi_UDI08;	
	
	eBuildingMode				: E_BA_BuildingMode;
	BuildingMode				: FB_BA_RawPublisher;
END_VAR

SUPER^(); // FB_BA_View
OpModMan(); // FB_BA_MV_Op
Sched(); // FB_BA_SchedM
DeMuxManMod(bEn := TRUE, nSel := OpModMan.nPresentValue, bIn := TRUE); // FB_BA_DMUX_B04
DeMuxSched(bEn := TRUE, nSel := Sched.nPresentValue, bIn := TRUE); // FB_BA_DMUX_B04
PrioSwi(
    bEn01 := DeMuxManMod.bQ02,
    nVal01 := E_BA_BuildingMode.eDefault,
    bEn02 := DeMuxManMod.bQ03,
    nVal02 := E_BA_BuildingMode.eNightWatch,
    bEn03 := DeMuxManMod.bQ04,
    nVal03 := E_BA_BuildingMode.eCleaning,
    bEn04 := FALSE,
    bEn05 := DeMuxSched.bQ01,
    nVal05 := E_BA_BuildingMode.eDefault,
    bEn06 := DeMuxSched.bQ02,
    nVal06 := E_BA_BuildingMode.eNightWatch,
    bEn07 := DeMuxSched.bQ03,
    nVal07 := E_BA_BuildingMode.eCleaning,
    bEn08 := FALSE); // FB_BA_PrioSwi_UDI08
OpModPr(nValuePgm := PrioSwi.nVal); // FB_BA_MV_Op
eBuildingMode := PrioSwi.nVal;
BuildingMode(xData := eBuildingMode); // FB_BA_RawPublisher

METHOD FB_init : BOOL
VAR_INPUT
	bInitRetains : BOOL; // if TRUE, the retain variables are initialized (warm start / cold start)
	bInCopyCode : BOOL;  // if TRUE, the instance afterwards gets moved into the copy code (online change)
END_VAR
OpModMan.iParent		:= THIS^;	
OpModMan.iLabel			:= LblCmpGeneral.BuildingMode_OpModMan;									
OpModMan.sObjectName	:= '{Idx=01}';
OpModMan.aStateText[1]	:= txtEvent_Auto;
OpModMan.aStateText[2]	:= txtEvent_Default;
OpModMan.aStateText[3]	:= txtEvent_Nightwatch;
OpModMan.aStateText[4]	:= txtEvent_Cleaning;
OpModMan.nValueRm		:= 1;

OpModPr.iParent			:= THIS^;	
OpModPr.iLabel			:= LblCmpGeneral.BuildingMode_OpModPr;									
OpModPr.sObjectName		:= '{Idx=01}';
OpModPr.aStateText[1]	:= txtEvent_Default;
OpModPr.aStateText[2]	:= txtEvent_Nightwatch;
OpModPr.aStateText[3]	:= txtEvent_Cleaning;
OpModPr.nValueRm		:= 1; 		
                        
Sched.iParent			:= THIS^;	
Sched.iLabel			:= LblCmpGeneral.BuildingMode_Sched;									
Sched.sObjectName		:= '{Idx=01}';
Sched.aStateText[1]		:= txtEvent_Default;
Sched.aStateText[2]		:= txtEvent_Nightwatch;
Sched.aStateText[3]		:= txtEvent_Cleaning;
Sched.nPredictTime		:= 0;


Sched.aWeek		:= F_BA_SchedWeekly4xM(E_BA_WeekDay.eMonday, E_BA_WeekDay.eFriday, T#0H, E_BA_BuildingMode.eNightWatch, T#6H, E_BA_BuildingMode.eDefault, T#19H, E_BA_BuildingMode.eCleaning, T#20H, E_BA_BuildingMode.eNightWatch);

(* alternatively
Sched.nDefaultValue										:= E_BA_BuildingMode.eDefault;
Sched.bWriteWeekly										:= FALSE;
//	Monday
Sched.aWeek[E_BA_Weekday.eMonday,1].eState				:= E_BA_SchedEntryState.eValue;
Sched.aWeek[E_BA_Weekday.eMonday,1].uValue.udiVal		:= E_BA_BuildingMode.eCleaning;
Sched.aWeek[E_BA_Weekday.eMonday,1].stTime.nHour		:= 19;
Sched.aWeek[E_BA_Weekday.eMonday,1].stTime.nMinute		:= 0;
Sched.aWeek[E_BA_Weekday.eMonday,1].stTime.nSecond		:= 0;
Sched.aWeek[E_BA_Weekday.eMonday,2].eState				:= E_BA_SchedEntryState.eValue;
Sched.aWeek[E_BA_Weekday.eMonday,2].uValue.udiVal		:= E_BA_BuildingMode.eNightWatch;
Sched.aWeek[E_BA_Weekday.eMonday,2].stTime.nHour		:= 20;
Sched.aWeek[E_BA_Weekday.eMonday,2].stTime.nMinute		:= 0;
Sched.aWeek[E_BA_Weekday.eMonday,2].stTime.nSecond		:= 0;
Sched.aWeek[E_BA_Weekday.eMonday,3].eState				:= E_BA_SchedEntryState.eValue;
Sched.aWeek[E_BA_Weekday.eMonday,3].uValue.udiVal		:= E_BA_BuildingMode.eDefault;
Sched.aWeek[E_BA_Weekday.eMonday,3].stTime.nHour		:= 0;
Sched.aWeek[E_BA_Weekday.eMonday,3].stTime.nMinute		:= 0;
Sched.aWeek[E_BA_Weekday.eMonday,3].stTime.nSecond		:= 0;
//	Tuesday
Sched.aWeek[E_BA_Weekday.eTuesday,1].eState				:= E_BA_SchedEntryState.eValue;
Sched.aWeek[E_BA_Weekday.eTuesday,1].uValue.udiVal		:= E_BA_BuildingMode.eCleaning;
Sched.aWeek[E_BA_Weekday.eTuesday,1].stTime.nHour		:= 19;
Sched.aWeek[E_BA_Weekday.eTuesday,1].stTime.nMinute		:= 0;
Sched.aWeek[E_BA_Weekday.eTuesday,1].stTime.nSecond		:= 0;
Sched.aWeek[E_BA_Weekday.eTuesday,2].eState				:= E_BA_SchedEntryState.eValue;
Sched.aWeek[E_BA_Weekday.eTuesday,2].uValue.udiVal		:= E_BA_BuildingMode.eNightWatch;
Sched.aWeek[E_BA_Weekday.eTuesday,2].stTime.nHour		:= 20;
Sched.aWeek[E_BA_Weekday.eTuesday,2].stTime.nMinute		:= 0;
Sched.aWeek[E_BA_Weekday.eTuesday,2].stTime.nSecond		:= 0;
Sched.aWeek[E_BA_Weekday.eTuesday,3].eState				:= E_BA_SchedEntryState.eValue;
Sched.aWeek[E_BA_Weekday.eTuesday,3].uValue.udiVal		:= E_BA_BuildingMode.eDefault;
Sched.aWeek[E_BA_Weekday.eTuesday,3].stTime.nHour		:= 0;
Sched.aWeek[E_BA_Weekday.eTuesday,3].stTime.nMinute		:= 0;
Sched.aWeek[E_BA_Weekday.eTuesday,3].stTime.nSecond		:= 0;
//	Wednesday
Sched.aWeek[E_BA_Weekday.eWednesday,1].eState			:= E_BA_SchedEntryState.eValue;
Sched.aWeek[E_BA_Weekday.eWednesday,1].uValue.udiVal	:= E_BA_BuildingMode.eCleaning;
Sched.aWeek[E_BA_Weekday.eWednesday,1].stTime.nHour		:= 19;
Sched.aWeek[E_BA_Weekday.eWednesday,1].stTime.nMinute	:= 0;
Sched.aWeek[E_BA_Weekday.eWednesday,1].stTime.nSecond	:= 0;
Sched.aWeek[E_BA_Weekday.eWednesday,2].eState			:= E_BA_SchedEntryState.eValue;
Sched.aWeek[E_BA_Weekday.eWednesday,2].uValue.udiVal	:= E_BA_BuildingMode.eNightWatch;
Sched.aWeek[E_BA_Weekday.eWednesday,2].stTime.nHour		:= 20;
Sched.aWeek[E_BA_Weekday.eWednesday,2].stTime.nMinute	:= 0;
Sched.aWeek[E_BA_Weekday.eWednesday,2].stTime.nSecond	:= 0;
Sched.aWeek[E_BA_Weekday.eWednesday,3].eState			:= E_BA_SchedEntryState.eValue;
Sched.aWeek[E_BA_Weekday.eWednesday,3].uValue.udiVal	:= E_BA_BuildingMode.eDefault;
Sched.aWeek[E_BA_Weekday.eWednesday,3].stTime.nHour		:= 0;
Sched.aWeek[E_BA_Weekday.eWednesday,3].stTime.nMinute	:= 0;
Sched.aWeek[E_BA_Weekday.eWednesday,3].stTime.nSecond	:= 0;
//	Thursday
Sched.aWeek[E_BA_Weekday.eThursday,1].eState			:= E_BA_SchedEntryState.eValue;
Sched.aWeek[E_BA_Weekday.eThursday,1].uValue.udiVal		:=E_BA_BuildingMode.eCleaning;
Sched.aWeek[E_BA_Weekday.eThursday,1].stTime.nHour		:= 19;
Sched.aWeek[E_BA_Weekday.eThursday,1].stTime.nMinute	:= 0;
Sched.aWeek[E_BA_Weekday.eThursday,1].stTime.nSecond	:= 0;
Sched.aWeek[E_BA_Weekday.eThursday,2].eState			:= E_BA_SchedEntryState.eValue;
Sched.aWeek[E_BA_Weekday.eThursday,2].uValue.udiVal		:= E_BA_BuildingMode.eNightWatch;
Sched.aWeek[E_BA_Weekday.eThursday,2].stTime.nHour		:= 20;
Sched.aWeek[E_BA_Weekday.eThursday,2].stTime.nMinute	:= 0;
Sched.aWeek[E_BA_Weekday.eThursday,2].stTime.nSecond	:= 0;
Sched.aWeek[E_BA_Weekday.eThursday,3].eState			:= E_BA_SchedEntryState.eValue;
Sched.aWeek[E_BA_Weekday.eThursday,3].uValue.udiVal		:= E_BA_BuildingMode.eDefault;
Sched.aWeek[E_BA_Weekday.eThursday,3].stTime.nHour		:= 0;
Sched.aWeek[E_BA_Weekday.eThursday,3].stTime.nMinute	:= 0;
Sched.aWeek[E_BA_Weekday.eThursday,3].stTime.nSecond	:= 0;
//	Friday
Sched.aWeek[E_BA_Weekday.eFriday,1].eState				:= E_BA_SchedEntryState.eValue;
Sched.aWeek[E_BA_Weekday.eFriday,1].uValue.udiVal		:= E_BA_BuildingMode.eCleaning;
Sched.aWeek[E_BA_Weekday.eFriday,1].stTime.nHour		:= 19;
Sched.aWeek[E_BA_Weekday.eFriday,1].stTime.nMinute		:= 0;
Sched.aWeek[E_BA_Weekday.eFriday,1].stTime.nSecond		:= 0;
Sched.aWeek[E_BA_Weekday.eFriday,2].eState				:= E_BA_SchedEntryState.eValue;
Sched.aWeek[E_BA_Weekday.eFriday,2].uValue.udiVal		:= E_BA_BuildingMode.eNightWatch;
Sched.aWeek[E_BA_Weekday.eFriday,2].stTime.nHour		:= 20;
Sched.aWeek[E_BA_Weekday.eFriday,2].stTime.nMinute		:= 0;
Sched.aWeek[E_BA_Weekday.eFriday,2].stTime.nSecond		:= 0;
Sched.aWeek[E_BA_Weekday.eFriday,3].eState				:= E_BA_SchedEntryState.eValue;
Sched.aWeek[E_BA_Weekday.eFriday,3].uValue.udiVal		:= E_BA_BuildingMode.eDefault;
Sched.aWeek[E_BA_Weekday.eFriday,3].stTime.nHour		:= 0;
Sched.aWeek[E_BA_Weekday.eFriday,3].stTime.nMinute		:= 0;
Sched.aWeek[E_BA_Weekday.eFriday,3].stTime.nSecond		:= 0; 
*)
END_METHOD

END_FUNCTION_BLOCK

// ---- Templates/POUs/Trade/AC/FB_BA_AC.TcPOU
{region '#Template'}
	{attribute 'Version' := '1.2.1.0'}
	{attribute 'Tags' := '"LCID": "1031", "Text": "Trade, Plant, AC"'}
	{attribute 'Tags' := '"LCID": "1033", "Text": "Trade, Plant, AC"'}
	{attribute 'Using' := '"Type": "Template", "URI": "Site"'}
	{attribute 'Description' := '"LCID": "1031", "Text": "Aufruf der Anlagen des Gewerks Klimaanlagen"'}
	{attribute 'Description' := '"LCID": "1033", "Text": "Calling the plants of the trade air conditioning"'}
{endregion}
FUNCTION_BLOCK FB_BA_AC EXTENDS FB_BA_View
VAR_INPUT CONSTANT
	AHU01				: FB_BA_AHU_1st_10;	
END_VAR
VAR_INPUT
END_VAR
VAR_OUTPUT
END_VAR
VAR
END_VAR

SUPER^(); // FB_BA_View
AHU01(); // FB_BA_AHU_1st_10

METHOD FB_init : BOOL
VAR_INPUT
	bInitRetains : BOOL; // if TRUE, the retain variables are initialized (warm start / cold start)
	bInCopyCode : BOOL;  // if TRUE, the instance afterwards gets moved into the copy code (online change)
END_VAR
AHU01.iParent 				:= THIS^;	
AHU01.sObjectName				:= '{PAC01}';											
AHU01.sDescription			:= '{Partial air-conditioning system}';							
AHU01.eDPADMode				:= E_BA_DPADMode.eInclude;

AHU01.GeneralSettings.Subject	:= Site.GeneralSettings_Subject;
AHU01.GeneralSettings.sTarget	:= Site.GeneralSettings_NetId;
END_METHOD

END_FUNCTION_BLOCK

// ---- Templates/POUs/Trade/AC/Plants/FB_BA_AHU_1st_10.TcPOU
{region '#Template'}
	{attribute 'Version' := '2.0.2.0'}
	{attribute 'Tags' := '"LCID": "1031", "Text": "AC, Plant, AHU, Lüftungsanlage"'}
	{attribute 'Tags' := '"LCID": "1033", "Text": "AC, Plant, AHU, Air handling unit"'}
	{attribute 'Using' := '"Type": "Template", "URI": "Site"'}
	{attribute 'Using' := '"Type": "Template", "URI": "E_BA_AC_OpMod01"'}
	{attribute 'Using' := '"Type": "Template", "URI": "E_BA_MdltCmd"'}
	{attribute 'Description' := '"LCID": "1031", "Text": "Ventilator druckgesteuert, Einfache Abluft/Zuluftkaskade, Vorerhitzer, ERC Platte, Kühler "'}
	{attribute 'Description' := '"LCID": "1033", "Text": "Fan pressure controlled, Simple extract air/supply air cascade, PreHeater, ERC Plate, Cooler"'}
{endregion}
FUNCTION_BLOCK FB_BA_AHU_1st_10 EXTENDS FB_BA_View
VAR_INPUT CONSTANT	
	TOuA					: FB_BA_SensorAnalog_IO;			
	TExhA					: FB_BA_SensorAnalog_IO;	
	TSuA					: FB_BA_SensorAnalog_IO;	
	TExtA					: FB_BA_SensorAnalog_IO;								
	TRm						: FB_BA_SensorAnalog_IO;	
	DiffPrssOuAFilt			: FB_BA_SensorAnalog_IO;											
	FiltOuAMonit			: FB_BA_Hys_21;							
	DiffPrssExtAFilt		: FB_BA_SensorAnalog_IO;				
	FiltExtAMonit			: FB_BA_Hys_21;	
	SumNgtCol				: FB_BA_AC_SumNgtCol;	
	OpMod					: FB_BA_AC_OpMod1St;	
	OuADmp					: FB_BA_Dmp2P;	
	SuAPrss					: FB_BA_SensorAnalog_IO;	
	SuADiffPrss				: FB_BA_SensorAnalog_IO;		
	SuAFan					: FB_BA_MotCtlExt;	
	SuADiffPrssMonit		: FB_BA_FdbAnalog;								
	ExhADmp					: FB_BA_Dmp2P;	
	ExtAPrss				: FB_BA_SensorAnalog_IO;	
	ExtADiffPrss			: FB_BA_SensorAnalog_IO;		
	ExtAFan					: FB_BA_MotCtlExt;								
	ExtADiffPrssMonit		: FB_BA_FdbAnalog;
	SpTRm					: FB_BA_Scale_04_Y2_3;	
	TCasCtrl				: FB_BA_AC_TCasCtrl_01;										 								
	TSeqLink				: FB_BA_SequenceLink;
	PreHtr					: FB_BA_AC_PreHtr;	
	Erc						: FB_BA_AC_ErcPl_02;								
	Col						: FB_BA_AC_ColT_02;								
	PlantCtrl				: FB_BA_PlantCtrl;							
	GeneralSettings			: FB_BA_RawSubscriber;
	stGeneralSettings		: ST_BA_GeneralSettings;
END_VAR	
VAR
	PlantLock				: FB_BA_PlantLock	:= (iParent := THIS^);	
	
	PlantControlStatus   	:FB_BA_Label2x :=(iAggregate:=LblControl_PlantControl,		iFunction:=LblFunctions_Status);
	TSequenceControlStatus  :FB_BA_Label2x :=(iAggregate:=LblControl_TSequenceControl,	iFunction:=LblFunctions_Status);	
END_VAR
VAR // added by the converter: edge detectors and wires of the graphical bodies
    _w1 : ANY;
END_VAR

SUPER^(); // FB_BA_View
GeneralSettings(xData := stGeneralSettings); // FB_BA_RawSubscriber
TOuA(); // FB_BA_SensorAnalog_IO
TSuA(); // FB_BA_SensorAnalog_IO
TExtA(); // FB_BA_SensorAnalog_IO
TExhA(); // FB_BA_SensorAnalog_IO
TRm(); // FB_BA_SensorAnalog_IO
DiffPrssOuAFilt(); // FB_BA_SensorAnalog_IO
DiffPrssExtAFilt(); // FB_BA_SensorAnalog_IO
FiltOuAMonit(bEn := TCasCtrl.bOn, fIn := DiffPrssOuAFilt.fPresentValue); // FB_BA_Hys_21
FiltExtAMonit(bEn := TCasCtrl.bOn, fIn := DiffPrssExtAFilt.fPresentValue); // FB_BA_Hys_21
SuAPrss(); // FB_BA_SensorAnalog_IO
SuADiffPrss(); // FB_BA_SensorAnalog_IO
OuADmp(bEnCrit := SuAFan.bOpState, bValCrit := TRUE); // FB_BA_Dmp2P
SuAFan(bEnCrit := NOT OuADmp.bSwiOpn, bValCrit := FALSE, fIn := SuAPrss.fPresentValue); // FB_BA_MotCtlExt
SuADiffPrssMonit(bEn := TCasCtrl.bOn, bCommand := SuAFan.bCmd, fIn := SuADiffPrss.fPresentValue); // FB_BA_FdbAnalog
ExtAPrss(); // FB_BA_SensorAnalog_IO
ExtADiffPrss(); // FB_BA_SensorAnalog_IO
ExhADmp(bEnCrit := ExtAFan.bOpState, bValCrit := TRUE); // FB_BA_Dmp2P
ExtAFan(bEnCrit := NOT ExhADmp.bSwiOpn, bValCrit := FALSE, fIn := ExtAPrss.fPresentValue); // FB_BA_MotCtlExt
ExtADiffPrssMonit(bEn := TCasCtrl.bOn, bCommand := ExtAFan.bCmd, fIn := ExtADiffPrss.fPresentValue); // FB_BA_FdbAnalog
PreHtr(
    fSpTSuA := TCasCtrl.fSpHtg,
    fTSuA := TSuA.fPresentValue,
    bDehumf := FALSE,
    bMixADmpAvail := FALSE,
    fTWth := stGeneralSettings.fTWth,
    bTWthLowLimit := stGeneralSettings.bTWthLowLimit); // FB_BA_AC_PreHtr
Erc(
    fSpTSuA := TCasCtrl.fSpErc,
    fTSuA := TSuA.fPresentValue,
    fTExhA := TExhA.fPresentValue,
    fTExtA := TExtA.fPresentValue,
    fTWth := stGeneralSettings.fTWth); // FB_BA_AC_ErcPl_02
Col(fSpTSuA := TCasCtrl.fSpCol, fTSuA := TSuA.fPresentValue); // FB_BA_AC_ColT_02
SpTRm(fTWth := stGeneralSettings.fTWth); // FB_BA_Scale_04_Y2_3
TCasCtrl(fSpTRm := SpTRm.fY, fTRm := TRm.fPresentValue); // FB_BA_AC_TCasCtrl_01
TSeqLink(bEn := TCasCtrl.bOn); // FB_BA_SequenceLink
PlantLock(); // FB_BA_PlantLock
_w1 := PlantLock.bPrioHigh OR PlantLock.bPrioMedium;
SumNgtCol(fTRm := TRm.fPresentValue, fSpRm := SpTRm.fY, fTWth := stGeneralSettings.fTWth); // FB_BA_AC_SumNgtCol
OpMod(bFrst := PreHtr.bFrost, bAlmShutOff := _w1, bNgtCol := SumNgtCol.bQ); // FB_BA_AC_OpMod1St
PlantCtrl(nOpMode := OpMod.eOpMode); // FB_BA_PlantCtrl

METHOD FB_init : BOOL
VAR_INPUT
	bInitRetains : BOOL; // if TRUE, the retain variables are initialized (warm start / cold start)
	bInCopyCode : BOOL;  // if TRUE, the instance afterwards gets moved into the copy code (online change)
END_VAR
GeneralSettings.Subject						:= Site.GeneralSettings_Subject;
GeneralSettings.sTarget						:= Site.GeneralSettings_NetId;		

TOuA.iParent								:= THIS^;		
TOuA.iLabel 								:= LblCmpAC.AHU_TOuA;	
TOuA.sObjectName							:= '{Idx=01}';	
TOuA.eDPADMode								:= E_BA_DPADMode.eInclude;										
TOuA.MV.eUnit								:= E_BA_Unit.eTemperature_DegreesCelsius;
TOuA.MV.fResolution 						:= 0.01;
TOuA.MV.fScaleOffset 						:= 0; 
TOuA.MV.bEventDetectionEnable				:= TRUE;
TOuA.MV.eEnPlantLock						:= E_BA_LockPriority.eNoLock;

TExhA.iParent								:= THIS^;		
TExhA.iLabel 								:= LblCmpAC.AHU_TExhA;	
TExhA.sObjectName							:= '{Idx=01}';												
TExhA.eDPADMode								:= E_BA_DPADMode.eInclude;										
TExhA.MV.eUnit								:= E_BA_Unit.eTemperature_DegreesCelsius;
TExhA.MV.fResolution 						:= 0.01;
TExhA.MV.fScaleOffset 						:= 0; 
TOuA.MV.bEventDetectionEnable				:= TRUE;
TOuA.MV.eEnPlantLock						:= E_BA_LockPriority.eNoLock;

TSuA.iParent								:= THIS^;		
TSuA.iLabel 								:= LblCmpAC.AHU_TSuA;	
TSuA.sObjectName							:= '{Idx=01}';
TSuA.eDPADMode								:= E_BA_DPADMode.eInclude;										
TSuA.MV.eUnit								:= E_BA_Unit.eTemperature_DegreesCelsius;
TSuA.MV.fResolution 						:= 0.01;
TSuA.MV.fScaleOffset 						:= 0; 
TSuA.MV.bEventDetectionEnable				:= TRUE;
TSuA.MV.eEnPlantLock						:= E_BA_LockPriority.eMedium;

TExtA.iParent								:= THIS^;
TExtA.iLabel 								:= LblCmpAC.AHU_TExtA;	
TExtA.sObjectName							:= '{Idx=01}'; 
TExtA.eDPADMode								:= E_BA_DPADMode.eInclude;										
TExtA.MV.eUnit								:= E_BA_Unit.eTemperature_DegreesCelsius;
TExtA.MV.fResolution 						:= 0.01;
TExtA.MV.fScaleOffset 						:= 0; 
TExtA.MV.bEventDetectionEnable				:= TRUE;
TExtA.MV.eEnPlantLock						:= E_BA_LockPriority.eNoLock;

TRm.iParent									:= THIS^;		
TRm.iLabel 									:= LblCmpAC.AHU_TRm;	
TRm.sObjectName								:= '{Idx=01}';
TRm.eDPADMode								:= E_BA_DPADMode.eInclude;										
TRm.MV.eUnit								:= E_BA_Unit.eTemperature_DegreesCelsius;
TRm.MV.fResolution 							:= 0.01;
TRm.MV.fScaleOffset 						:= 0;
TRm.MV.bEventDetectionEnable				:= TRUE;
TRm.MV.eEnPlantLock							:= E_BA_LockPriority.eNoLock;

DiffPrssOuAFilt.iParent								:= THIS^;		
DiffPrssOuAFilt.iLabel 								:= LblCmpAC.AHU_DiffPrssOuAFilt;	
DiffPrssOuAFilt.sObjectName							:= '{Idx=03}';												
DiffPrssOuAFilt.eDPADMode							:= E_BA_DPADMode.eInclude;										
DiffPrssOuAFilt.MV.eUnit							:= E_BA_Unit.ePressure_Pascals;
DiffPrssOuAFilt.MV.fResolution 						:= 0.03051851;
DiffPrssOuAFilt.MV.fScaleOffset 					:= 0; 
DiffPrssOuAFilt.MV.bEventDetectionEnable			:= TRUE;
DiffPrssOuAFilt.MV.eEnPlantLock						:= E_BA_LockPriority.eNoLock;

FiltOuAMonit.iParent								:= THIS^;
FiltOuAMonit.iLabel									:= LblCmpAC.AHU_FiltOuAMonit;
FiltOuAMonit.sObjectName							:= '{Idx=01}';										 
FiltOuAMonit.eDPADMode								:= E_BA_DPADMode.eInclude;
FiltOuAMonit.DstPreAlarm.bEventDetectionEnable		:= TRUE;
FiltOuAMonit.DstPreAlarm.eEnPlantLock				:= E_BA_LockPriority.eNoLock;	
FiltOuAMonit.DstMainAlarm.bEventDetectionEnable		:= TRUE;
FiltOuAMonit.DstMainAlarm.eEnPlantLock				:= E_BA_LockPriority.eMedium;

DiffPrssExtAFilt.iParent							:= THIS^;		
DiffPrssExtAFilt.iLabel 							:= LblCmpAC.AHU_DiffPrssExtAFilt;	
DiffPrssExtAFilt.sObjectName						:= '{Idx=04}';
DiffPrssExtAFilt.eDPADMode							:= E_BA_DPADMode.eInclude;										
DiffPrssExtAFilt.MV.eUnit							:= E_BA_Unit.ePressure_Pascals;
DiffPrssExtAFilt.MV.fResolution 					:= 0.03051851;
DiffPrssExtAFilt.MV.fScaleOffset 					:= 0; 
DiffPrssExtAFilt.MV.bEventDetectionEnable			:= TRUE;
DiffPrssExtAFilt.MV.eEnPlantLock					:= E_BA_LockPriority.eNoLock;

FiltExtAMonit.iParent								:= THIS^;
FiltExtAMonit.iLabel								:= LblCmpAC.AHU_FiltExtAMonit;
FiltExtAMonit.sObjectName							:= '{Idx=02}';										 
FiltExtAMonit.eDPADMode								:= E_BA_DPADMode.eInclude;
FiltExtAMonit.DstPreAlarm.bEventDetectionEnable		:= TRUE;
FiltExtAMonit.DstPreAlarm.eEnPlantLock				:= E_BA_LockPriority.eNoLock;	
FiltExtAMonit.DstMainAlarm.bEventDetectionEnable	:= TRUE;
FiltExtAMonit.DstMainAlarm.eEnPlantLock				:= E_BA_LockPriority.eMedium;

SumNgtCol.iParent							:= THIS^;
SumNgtCol.iLabel							:= LblCmpAC.AHU_SumNgtCol;
SumNgtCol.sObjectName						:= '{Idx=01}';										 
SumNgtCol.eDPADMode							:= E_BA_DPADMode.eInclude;								

OpMod.iParent								:= THIS^;
OpMod.iLabel								:= LblCmpAC.AHU_OpMod;
OpMod.sObjectName							:= '{Idx=01}';										 
OpMod.eDPADMode								:= E_BA_DPADMode.eInclude;								

OuADmp.iParent								:= THIS^;
OuADmp.iLabel								:= LblCmpAC.AHU_OuADmp;
OuADmp.sObjectName							:= '{Idx=01}';										 
OuADmp.eDPADMode							:= E_BA_DPADMode.eInclude;
OuADmp.MonitOpen.Dst.eEnPlantLock			:= E_BA_LockPriority.eLocalMedium;
OuADmp.MonitOpen.Dst.bEventDetectionEnable	:= TRUE;						
OuADmp.MonitClose.Dst.eEnPlantLock			:= E_BA_LockPriority.eNoLock;								
OuADmp.MonitClose.Dst.bEventDetectionEnable	:= TRUE;						

SuAPrss.iParent								:= THIS^;		
SuAPrss.iLabel 								:= LblCmpAC.AHU_SuAPrss;	
SuAPrss.sObjectName							:= '{Idx=01}';
SuAPrss.eDPADMode							:= E_BA_DPADMode.eInclude;																						
SuAPrss.MV.eUnit							:= E_BA_Unit.ePressure_Pascals;
SuAPrss.MV.fResolution 						:= 0.03051851;
SuAPrss.MV.fScaleOffset 					:= 0;
SuAPrss.MV.bEventDetectionEnable			:= TRUE;
SuAPrss.MV.eEnPlantLock						:= E_BA_LockPriority.eNoLock;

SuADiffPrss.iParent							:= THIS^;		
SuADiffPrss.iLabel 							:= LblCmpAC.AHU_SuADiffPrss;	
SuADiffPrss.sObjectName						:= '{Idx=01}';
SuADiffPrss.eDPADMode						:= E_BA_DPADMode.eInclude;																						
SuADiffPrss.MV.eUnit						:= E_BA_Unit.ePressure_Pascals;
SuADiffPrss.MV.fResolution 					:= 0.03051851;
SuADiffPrss.MV.fScaleOffset 				:= 0; 
SuADiffPrss.MV.bEventDetectionEnable		:= TRUE;
SuADiffPrss.MV.eEnPlantLock					:= E_BA_LockPriority.eNoLock;

SuAFan.iParent								:= THIS^;
SuAFan.iLabel								:= LblCmpAC.AHU_SuAFan;
SuAFan.sObjectName							:= '{Idx=01}';										 
SuAFan.eDPADMode							:= E_BA_DPADMode.eInclude;								
SuAFan.Dst.eEnPlantLock						:= E_BA_LockPriority.eMedium;
SuAFan.Dst.bEventDetectionEnable			:= TRUE;
SuAFan.ThOvrld.eEnPlantLock					:= E_BA_LockPriority.eMedium;	
SuAFan.ThOvrld.bEventDetectionEnable		:= TRUE;
SuAFan.MntnSwi.eEnPlantLock					:= E_BA_LockPriority.eMedium;
SuAFan.MntnSwi.bEventDetectionEnable		:= TRUE;

SuADiffPrssMonit.iParent					:= THIS^;
SuADiffPrssMonit.iLabel						:= LblCmpAC.AHU_SuADiffPrssMonit;
SuADiffPrssMonit.sObjectName				:= '{Idx=01}';										 
SuADiffPrssMonit.eDPADMode					:= E_BA_DPADMode.eInclude;
SuADiffPrssMonit.Dst.bEventDetectionEnable	:= TRUE;								
SuADiffPrssMonit.Dst.eEnPlantLock			:= E_BA_LockPriority.eMedium;				

ExhADmp.iParent								:= THIS^;
ExhADmp.iLabel								:= LblCmpAC.AHU_ExhADmp;
ExhADmp.sObjectName							:= '{Idx=02}';										 
ExhADmp.eDPADMode							:= E_BA_DPADMode.eInclude;								
ExhADmp.MonitOpen.Dst.eEnPlantLock			:= E_BA_LockPriority.eLocalMedium;								
ExhADmp.MonitOpen.Dst.bEventDetectionEnable	:= TRUE;						
ExhADmp.MonitClose.Dst.eEnPlantLock			:= E_BA_LockPriority.eNoLock;				
ExhADmp.MonitClose.Dst.bEventDetectionEnable:= TRUE;	

ExtAPrss.iParent							:= THIS^;		
ExtAPrss.iLabel 							:= LblCmpAC.AHU_ExtAPrss;	
ExtAPrss.sObjectName						:= '{Idx=01}';												
ExtAPrss.eDPADMode							:= E_BA_DPADMode.eInclude;																						
ExtAPrss.MV.eUnit							:= E_BA_Unit.ePressure_Pascals;
ExtAPrss.MV.fResolution 					:= 0.03051851;
ExtAPrss.MV.fScaleOffset 					:= 0; 
ExtAPrss.MV.bEventDetectionEnable			:= TRUE;
ExtAPrss.MV.eEnPlantLock					:= E_BA_LockPriority.eNoLock;

ExtADiffPrss.iParent						:= THIS^;		
ExtADiffPrss.iLabel 						:= LblCmpAC.AHU_ExtADiffPrss;	
ExtADiffPrss.sObjectName					:= '{Idx=02}';
ExtADiffPrss.eDPADMode						:= E_BA_DPADMode.eInclude;																						
ExtADiffPrss.MV.eUnit						:= E_BA_Unit.ePressure_Pascals;
ExtADiffPrss.MV.fResolution 				:= 0.03051851;
ExtADiffPrss.MV.fScaleOffset 				:= 0; 
ExtADiffPrss.MV.bEventDetectionEnable		:= TRUE;
ExtADiffPrss.MV.eEnPlantLock				:= E_BA_LockPriority.eNoLock;

ExtAFan.iParent								:= THIS^;
ExtAFan.iLabel								:= LblCmpAC.AHU_ExtAFan;
ExtAFan.sObjectName							:= '{Idx=01}';										 
ExtAFan.eDPADMode							:= E_BA_DPADMode.eInclude;								
ExtAFan.Dst.eEnPlantLock					:= E_BA_LockPriority.eMedium;
ExtAFan.Dst.bEventDetectionEnable			:= TRUE;
ExtAFan.ThOvrld.eEnPlantLock				:= E_BA_LockPriority.eMedium;	
ExtAFan.ThOvrld.bEventDetectionEnable		:= TRUE;
ExtAFan.MntnSwi.eEnPlantLock				:= E_BA_LockPriority.eMedium;
ExtAFan.MntnSwi.bEventDetectionEnable		:= TRUE;

ExtADiffPrssMonit.iParent					:= THIS^;
ExtADiffPrssMonit.iLabel					:= LblCmpAC.AHU_ExtADiffPrssMonit;
ExtADiffPrssMonit.sObjectName				:= '{Idx=02}';										 
ExtADiffPrssMonit.eDPADMode					:= E_BA_DPADMode.eInclude;								
ExtADiffPrssMonit.Dst.bEventDetectionEnable	:= TRUE;										
ExtADiffPrssMonit.Dst.eEnPlantLock			:= E_BA_LockPriority.eMedium;													

SpTRm.iParent								:= THIS^;
SpTRm.iLabel								:= LblCmpAC.AHU_SpTRm;
SpTRm.sObjectName							:= '{Idx=01}';										 
SpTRm.eDPADMode								:= E_BA_DPADMode.eInclude;								

TCasCtrl.iParent							:= THIS^;
TCasCtrl.iLabel								:= LblCmpAC.AHU_TCasCtrl;
TCasCtrl.sObjectName						:= '{Idx=01}';										 
TCasCtrl.eDPADMode							:= E_BA_DPADMode.eInclude;																		 								

TSeqLink.iParent							:= THIS^;
TSeqLink.iLabel								:= LblCmpAC.AHU_TSeqLink;
TSeqLink.sObjectName						:= '{Idx=01,Idx=01}';									
TSeqLink.iReference[1]						:= PreHtr.TSuACtrl.Ctrl;
TSeqLink.iReference[2]						:= Erc.TSuACtrl.Ctrl;
TSeqLink.iReference[3]						:= Col.TSuACtrl.Ctrl;
TSeqLink.aStateText[1]						:= txtEvent_SupplyAirTControlPreheater;
TSeqLink.aStateText[2]						:= txtEvent_SupplyAirTControlERC;
TSeqLink.aStateText[3]						:= txtEvent_SupplyAirTControlCooler;
	
PreHtr.iParent										:= THIS^;
PreHtr.iLabel										:= LblCmpAC.AHU_PreHtr;
PreHtr.sObjectName									:= '{Idx=01}';										 
PreHtr.eDPADMode									:= E_BA_DPADMode.eIncludeDescription;								
PreHtr.TFl.MV.bEventDetectionEnable					:= TRUE;
PreHtr.TRt.MV.eEnPlantLock							:= E_BA_LockPriority.eMedium;
PreHtr.TRt.MV.bEventDetectionEnable					:= TRUE;
PreHtr.TRtCtrl.PreRinseDst.eEnPlantLock				:= E_BA_LockPriority.eNoLock;
PreHtr.TRtCtrl.PreRinseDst.bEventDetectionEnable	:= TRUE;
PreHtr.TFrost.MV.eEnPlantLock						:= E_BA_LockPriority.eMedium;
PreHtr.TFrost.MV.bEventDetectionEnable				:= TRUE;
PreHtr.FrostThermostat.Input.eEnPlantLock			:= E_BA_LockPriority.eMedium;	
PreHtr.FrostThermostat.Input.bEventDetectionEnable	:= TRUE;	
PreHtr.Pu.Dst.eEnPlantLock							:= E_BA_LockPriority.eMedium;
PreHtr.Pu.Dst.bEventDetectionEnable					:= TRUE;

Erc.iParent									:= THIS^;
Erc.iLabel									:= LblCmpAC.AHU_Erc;
Erc.sObjectName								:= '{Idx=01}';										 
Erc.eDPADMode								:= E_BA_DPADMode.eIncludeDescription;																
Erc.DiffPrssSwi.Input.bEventDetectionEnable	:= TRUE;

Col.iParent									:= THIS^;
Col.iLabel									:= LblCmpAC.AHU_Col;
Col.sObjectName								:= '{Idx=01}';										 
Col.eDPADMode								:= E_BA_DPADMode.eIncludeDescription;								
Col.TFl.MV.bEventDetectionEnable			:= TRUE;
Col.TRt.MV.bEventDetectionEnable			:= TRUE;	

PlantCtrl.iParent							:= THIS^;
PlantCtrl.iLabel							:= LblCmpAC.AHU_PlantCtrl;
PlantCtrl.sObjectName						:= '{Idx=01,Idx=01}';
//	PlantCtrl.aStateText						:= OpMod.OpModPr.aStateText;	

	
// Die folgenden Aufrufe müssen am Schluss aufgerufen sein!!! // The following calls must be called at the end!!!
PlantCtrl.Clear();
Init_OffOn();
END_METHOD

METHOD Init_OffOn : BOOL
// Betriebsarten der Anlage mit Prioritäten
// plant operations modes with priorities
PlantCtrl.AddOperationMode(nOpMode := E_BA_AC_OpMod01.eOff,							ePrio := E_BA_Priority.eProgram,		eIgnore := E_BA_AggregateIgnoreFlags.None);
PlantCtrl.AddOperationMode(nOpMode := E_BA_AC_OpMod01.eOn,							ePrio := E_BA_Priority.eProgram,		eIgnore := E_BA_AggregateIgnoreFlags.None);
PlantCtrl.AddOperationMode(nOpMode := E_BA_AC_OpMod01.eNightCooling,				ePrio := E_BA_Priority.eProgram,		eIgnore := E_BA_AggregateIgnoreFlags.None);
PlantCtrl.AddOperationMode(nOpMode := E_BA_AC_OpMod01.eCoolDownProtection,			ePrio := E_BA_Priority.eProgram,		eIgnore := E_BA_AggregateIgnoreFlags.None);
PlantCtrl.AddOperationMode(nOpMode := E_BA_AC_OpMod01.eOverHeatingProtection,		ePrio := E_BA_Priority.eProgram,		eIgnore := E_BA_AggregateIgnoreFlags.None);
PlantCtrl.AddOperationMode(nOpMode := E_BA_AC_OpMod01.eFrost,						ePrio := E_BA_Priority.eCritical,		eIgnore := E_BA_AggregateIgnoreFlags.None);
PlantCtrl.AddOperationMode(nOpMode := E_BA_AC_OpMod01.eEmergency,					ePrio := E_BA_Priority.eCritical,		eIgnore := E_BA_AggregateIgnoreFlags.None);
PlantCtrl.AddOperationMode(nOpMode := E_BA_AC_OpMod01.eAlarm,						ePrio := E_BA_Priority.eCritical,		eIgnore := E_BA_AggregateIgnoreFlags.None);
PlantCtrl.AddOperationMode(nOpMode := E_BA_AC_OpMod01.eForcedVentilation,			ePrio := E_BA_Priority.eCritical,		eIgnore := E_BA_AggregateIgnoreFlags.None);
PlantCtrl.AddOperationMode(nOpMode := E_BA_AC_OpMod01.eCentralSwitchOff,			ePrio := E_BA_Priority.eCritical,		eIgnore := E_BA_AggregateIgnoreFlags.None);
PlantCtrl.AddOperationMode(nOpMode := E_BA_AC_OpMod01.eSmokeExtractionProgramm,		ePrio := E_BA_Priority.eLifeSafety,		eIgnore := E_BA_AggregateIgnoreFlags.None);
PlantCtrl.AddOperationMode(nOpMode := E_BA_AC_OpMod01.eSmokeExtractionSupplyAir,	ePrio := E_BA_Priority.eLifeSafety,		eIgnore := E_BA_AggregateIgnoreFlags.None);
PlantCtrl.AddOperationMode(nOpMode := E_BA_AC_OpMod01.eSmokeExtractionExhaustAir,	ePrio := E_BA_Priority.eLifeSafety,		eIgnore := E_BA_AggregateIgnoreFlags.None);
PlantCtrl.AddOperationMode(nOpMode := E_BA_AC_OpMod01.eFire, 						ePrio := E_BA_Priority.eLifeSafety,		eIgnore := E_BA_AggregateIgnoreFlags.None);

// Startsequenz Schrittfolge und Parameter
// Start sequence Step order and parameter
PlantCtrl.AddAggregate(iRef := PreHtr,		bWaitForProcesses := TRUE,	bWaitForEvents := FALSE, tDelayStepDown := T#0S, tDelayStepUp := T#5S);
PlantCtrl.AddAggregate(iRef := OuADmp,		bWaitForProcesses := FALSE, bWaitForEvents := FALSE, tDelayStepDown := T#2S, tDelayStepUp := T#2S);
PlantCtrl.AddAggregate(iRef := ExhADmp,		bWaitForProcesses := FALSE, bWaitForEvents := FALSE, tDelayStepDown := T#2S, tDelayStepUp := T#2S);
PlantCtrl.AddAggregate(iRef := SuAFan,		bWaitForProcesses := FALSE, bWaitForEvents := FALSE, tDelayStepDown := T#2S, tDelayStepUp := T#2S);
PlantCtrl.AddAggregate(iRef := ExtAFan,		bWaitForProcesses := FALSE, bWaitForEvents := FALSE, tDelayStepDown := T#2S, tDelayStepUp := T#2S);
PlantCtrl.AddAggregate(iRef := Erc,			bWaitForProcesses := FALSE, bWaitForEvents := FALSE, tDelayStepDown := T#0S, tDelayStepUp := T#0S);
PlantCtrl.AddAggregate(iRef := Col,			bWaitForProcesses := FALSE, bWaitForEvents := FALSE, tDelayStepDown := T#0S, tDelayStepUp := T#0S);
PlantCtrl.AddAggregate(iRef := TCasCtrl,	bWaitForProcesses := FALSE, bWaitForEvents := FALSE, tDelayStepDown := T#0S, tDelayStepUp := T#0S);

// Aggregatbetriebsarten in Abhängigkeit von den entsprechenden Anlagenbetriebsarten anwenden
// Vorwärmer freigeben in Abhängigkeit von der Anlagenbetriebsart 
// Apply aggregate operation modes dependant on corresponding plant operation modes
// release pre-heater depending on plant operation mode 
PlantCtrl.AssignAggregate1x(nPltOpMode := E_BA_AC_OpMod01.eOff,							iAgg1Ref := PreHtr, nAgg1OpMode := TO_UDINT(FALSE));
PlantCtrl.AssignAggregate1x(nPltOpMode := E_BA_AC_OpMod01.eOn,							iAgg1Ref := PreHtr, nAgg1OpMode := TO_UDINT(TRUE));
PlantCtrl.AssignAggregate1x(nPltOpMode := E_BA_AC_OpMod01.eNightCooling,				iAgg1Ref := PreHtr, nAgg1OpMode := TO_UDINT(FALSE));
PlantCtrl.AssignAggregate1x(nPltOpMode := E_BA_AC_OpMod01.eCoolDownProtection,			iAgg1Ref := PreHtr, nAgg1OpMode := TO_UDINT(TRUE));
PlantCtrl.AssignAggregate1x(nPltOpMode := E_BA_AC_OpMod01.eOverHeatingProtection,		iAgg1Ref := PreHtr, nAgg1OpMode := TO_UDINT(FALSE));
PlantCtrl.AssignAggregate1x(nPltOpMode := E_BA_AC_OpMod01.eFrost,						iAgg1Ref := PreHtr, nAgg1OpMode := TO_UDINT(FALSE));
PlantCtrl.AssignAggregate1x(nPltOpMode := E_BA_AC_OpMod01.eEmergency,					iAgg1Ref := PreHtr, nAgg1OpMode := TO_UDINT(FALSE));
PlantCtrl.AssignAggregate1x(nPltOpMode := E_BA_AC_OpMod01.eAlarm,						iAgg1Ref := PreHtr, nAgg1OpMode := TO_UDINT(FALSE));
PlantCtrl.AssignAggregate1x(nPltOpMode := E_BA_AC_OpMod01.eForcedVentilation,			iAgg1Ref := PreHtr, nAgg1OpMode := TO_UDINT(TRUE));
PlantCtrl.AssignAggregate1x(nPltOpMode := E_BA_AC_OpMod01.eCentralSwitchOff,			iAgg1Ref := PreHtr, nAgg1OpMode := TO_UDINT(FALSE));
PlantCtrl.AssignAggregate1x(nPltOpMode := E_BA_AC_OpMod01.eSmokeExtractionProgramm,		iAgg1Ref := PreHtr, nAgg1OpMode := TO_UDINT(TRUE));
PlantCtrl.AssignAggregate1x(nPltOpMode := E_BA_AC_OpMod01.eSmokeExtractionSupplyAir,	iAgg1Ref := PreHtr, nAgg1OpMode := TO_UDINT(TRUE));
PlantCtrl.AssignAggregate1x(nPltOpMode := E_BA_AC_OpMod01.eSmokeExtractionExhaustAir,	iAgg1Ref := PreHtr, nAgg1OpMode := TO_UDINT(FALSE));
PlantCtrl.AssignAggregate1x(nPltOpMode := E_BA_AC_OpMod01.eFire,						iAgg1Ref := PreHtr, nAgg1OpMode := TO_UDINT(FALSE));

// Aggregatbetriebsarten in Abhängigkeit von den entsprechenden Anlagenbetriebsarten anwenden:
// Erc in Abhängigkeit von der Anlagenbetriebsart freigeben 
// Apply aggregate operation modes dependant on corresponding plant operation modes:
// release Erc depending on plant operation mode 
PlantCtrl.AssignAggregate1x(nPltOpMode := E_BA_AC_OpMod01.eOff,							iAgg1Ref := Erc, nAgg1OpMode := TO_UDINT(FALSE));
PlantCtrl.AssignAggregate1x(nPltOpMode := E_BA_AC_OpMod01.eOn,							iAgg1Ref := Erc, nAgg1OpMode := TO_UDINT(TRUE));
PlantCtrl.AssignAggregate1x(nPltOpMode := E_BA_AC_OpMod01.eNightCooling,				iAgg1Ref := Erc, nAgg1OpMode := TO_UDINT(FALSE));
PlantCtrl.AssignAggregate1x(nPltOpMode := E_BA_AC_OpMod01.eCoolDownProtection,			iAgg1Ref := Erc, nAgg1OpMode := TO_UDINT(TRUE));
PlantCtrl.AssignAggregate1x(nPltOpMode := E_BA_AC_OpMod01.eOverHeatingProtection,		iAgg1Ref := Erc, nAgg1OpMode := TO_UDINT(TRUE));
PlantCtrl.AssignAggregate1x(nPltOpMode := E_BA_AC_OpMod01.eFrost,						iAgg1Ref := Erc, nAgg1OpMode := TO_UDINT(FALSE));
PlantCtrl.AssignAggregate1x(nPltOpMode := E_BA_AC_OpMod01.eEmergency,					iAgg1Ref := Erc, nAgg1OpMode := TO_UDINT(FALSE));
PlantCtrl.AssignAggregate1x(nPltOpMode := E_BA_AC_OpMod01.eAlarm,						iAgg1Ref := Erc, nAgg1OpMode := TO_UDINT(FALSE));
PlantCtrl.AssignAggregate1x(nPltOpMode := E_BA_AC_OpMod01.eForcedVentilation,			iAgg1Ref := Erc, nAgg1OpMode := TO_UDINT(TRUE));
PlantCtrl.AssignAggregate1x(nPltOpMode := E_BA_AC_OpMod01.eCentralSwitchOff,			iAgg1Ref := Erc, nAgg1OpMode := TO_UDINT(FALSE));
PlantCtrl.AssignAggregate1x(nPltOpMode := E_BA_AC_OpMod01.eSmokeExtractionProgramm,		iAgg1Ref := Erc, nAgg1OpMode := TO_UDINT(TRUE));
PlantCtrl.AssignAggregate1x(nPltOpMode := E_BA_AC_OpMod01.eSmokeExtractionSupplyAir,	iAgg1Ref := Erc, nAgg1OpMode := TO_UDINT(TRUE));
PlantCtrl.AssignAggregate1x(nPltOpMode := E_BA_AC_OpMod01.eSmokeExtractionExhaustAir,	iAgg1Ref := Erc, nAgg1OpMode := TO_UDINT(TRUE));
PlantCtrl.AssignAggregate1x(nPltOpMode := E_BA_AC_OpMod01.eFire,						iAgg1Ref := Erc, nAgg1OpMode := TO_UDINT(FALSE));

// Aggregatbetriebsarten in Abhängigkeit von den entsprechenden Anlagenbetriebsarten anwenden:
// Kühler in Abhängigkeit von der Anlagenbetriebsart freigeben
// Apply aggregate operation modes dependant on corresponding plant operation modes:
// release cooler depending on plant operation mode 
PlantCtrl.AssignAggregate1x(nPltOpMode := E_BA_AC_OpMod01.eOff,							iAgg1Ref := Col, nAgg1OpMode := TO_UDINT(FALSE));
PlantCtrl.AssignAggregate1x(nPltOpMode := E_BA_AC_OpMod01.eOn,							iAgg1Ref := Col, nAgg1OpMode := TO_UDINT(TRUE));
PlantCtrl.AssignAggregate1x(nPltOpMode := E_BA_AC_OpMod01.eNightCooling,				iAgg1Ref := Col, nAgg1OpMode := TO_UDINT(FALSE));
PlantCtrl.AssignAggregate1x(nPltOpMode := E_BA_AC_OpMod01.eCoolDownProtection,			iAgg1Ref := Col, nAgg1OpMode := TO_UDINT(FALSE));
PlantCtrl.AssignAggregate1x(nPltOpMode := E_BA_AC_OpMod01.eOverHeatingProtection,		iAgg1Ref := Col, nAgg1OpMode := TO_UDINT(TRUE));
PlantCtrl.AssignAggregate1x(nPltOpMode := E_BA_AC_OpMod01.eFrost,						iAgg1Ref := Col, nAgg1OpMode := TO_UDINT(FALSE));
PlantCtrl.AssignAggregate1x(nPltOpMode := E_BA_AC_OpMod01.eEmergency,					iAgg1Ref := Col, nAgg1OpMode := TO_UDINT(FALSE));
PlantCtrl.AssignAggregate1x(nPltOpMode := E_BA_AC_OpMod01.eAlarm,						iAgg1Ref := Col, nAgg1OpMode := TO_UDINT(FALSE));
PlantCtrl.AssignAggregate1x(nPltOpMode := E_BA_AC_OpMod01.eForcedVentilation,			iAgg1Ref := Col, nAgg1OpMode := TO_UDINT(TRUE));
PlantCtrl.AssignAggregate1x(nPltOpMode := E_BA_AC_OpMod01.eCentralSwitchOff,			iAgg1Ref := Col, nAgg1OpMode := TO_UDINT(FALSE));
PlantCtrl.AssignAggregate1x(nPltOpMode := E_BA_AC_OpMod01.eSmokeExtractionProgramm,		iAgg1Ref := Col, nAgg1OpMode := TO_UDINT(FALSE));
PlantCtrl.AssignAggregate1x(nPltOpMode := E_BA_AC_OpMod01.eSmokeExtractionSupplyAir,	iAgg1Ref := Col, nAgg1OpMode := TO_UDINT(FALSE));
PlantCtrl.AssignAggregate1x(nPltOpMode := E_BA_AC_OpMod01.eSmokeExtractionExhaustAir,	iAgg1Ref := Col, nAgg1OpMode := TO_UDINT(FALSE));
PlantCtrl.AssignAggregate1x(nPltOpMode := E_BA_AC_OpMod01.eFire,						iAgg1Ref := Col, nAgg1OpMode := TO_UDINT(FALSE));

// Aggregatbetriebsarten in Abhängigkeit von den entsprechenden Anlagenbetriebsarten anwenden:
// Außenluftklappe freigeben in Abhängigkeit von der Anlagenbetriebsart 
// Apply aggregate operation modes dependant on corresponding plant operation modes:
// release outside air damper depending on plant operation mode 
PlantCtrl.AssignAggregate1x(nPltOpMode := E_BA_AC_OpMod01.eOff,							iAgg1Ref := OuADmp, nAgg1OpMode := TO_UDINT(FALSE));
PlantCtrl.AssignAggregate1x(nPltOpMode := E_BA_AC_OpMod01.eOn,							iAgg1Ref := OuADmp, nAgg1OpMode := TO_UDINT(TRUE));
PlantCtrl.AssignAggregate1x(nPltOpMode := E_BA_AC_OpMod01.eNightCooling,				iAgg1Ref := OuADmp, nAgg1OpMode := TO_UDINT(TRUE));
PlantCtrl.AssignAggregate1x(nPltOpMode := E_BA_AC_OpMod01.eCoolDownProtection,			iAgg1Ref := OuADmp, nAgg1OpMode := TO_UDINT(TRUE));
PlantCtrl.AssignAggregate1x(nPltOpMode := E_BA_AC_OpMod01.eOverHeatingProtection,		iAgg1Ref := OuADmp, nAgg1OpMode := TO_UDINT(TRUE));
PlantCtrl.AssignAggregate1x(nPltOpMode := E_BA_AC_OpMod01.eFrost,						iAgg1Ref := OuADmp, nAgg1OpMode := TO_UDINT(FALSE));
PlantCtrl.AssignAggregate1x(nPltOpMode := E_BA_AC_OpMod01.eEmergency,					iAgg1Ref := OuADmp, nAgg1OpMode := TO_UDINT(FALSE));
PlantCtrl.AssignAggregate1x(nPltOpMode := E_BA_AC_OpMod01.eAlarm,						iAgg1Ref := OuADmp, nAgg1OpMode := TO_UDINT(FALSE));
PlantCtrl.AssignAggregate1x(nPltOpMode := E_BA_AC_OpMod01.eForcedVentilation,			iAgg1Ref := OuADmp, nAgg1OpMode := TO_UDINT(TRUE));
PlantCtrl.AssignAggregate1x(nPltOpMode := E_BA_AC_OpMod01.eCentralSwitchOff,			iAgg1Ref := OuADmp, nAgg1OpMode := TO_UDINT(FALSE));
PlantCtrl.AssignAggregate1x(nPltOpMode := E_BA_AC_OpMod01.eSmokeExtractionProgramm,		iAgg1Ref := OuADmp, nAgg1OpMode := TO_UDINT(TRUE));
PlantCtrl.AssignAggregate1x(nPltOpMode := E_BA_AC_OpMod01.eSmokeExtractionSupplyAir,	iAgg1Ref := OuADmp, nAgg1OpMode := TO_UDINT(TRUE));
PlantCtrl.AssignAggregate1x(nPltOpMode := E_BA_AC_OpMod01.eSmokeExtractionExhaustAir,	iAgg1Ref := OuADmp, nAgg1OpMode := TO_UDINT(FALSE));
PlantCtrl.AssignAggregate1x(nPltOpMode := E_BA_AC_OpMod01.eFire,						iAgg1Ref := OuADmp, nAgg1OpMode := TO_UDINT(FALSE));

// Aggregatbetriebsarten in Abhängigkeit von den entsprechenden Anlagenbetriebsarten anwenden:
// Zuluftventilator freigeben in Abhängigkeit von der Anlagenbetriebsart 
// Apply aggregate operation modes dependant on corresponding plant operation modes:
// release supply air fan depending on plant operation mode 
PlantCtrl.AssignAggregate1x(nPltOpMode := E_BA_AC_OpMod01.eOff,							iAgg1Ref := SuAFan, nAgg1OpMode := E_BA_MdltCmd.eOff);
PlantCtrl.AssignAggregate1x(nPltOpMode := E_BA_AC_OpMod01.eOn,							iAgg1Ref := SuAFan, nAgg1OpMode := E_BA_MdltCmd.eOn);
PlantCtrl.AssignAggregate1x(nPltOpMode := E_BA_AC_OpMod01.eNightCooling,				iAgg1Ref := SuAFan, nAgg1OpMode := E_BA_MdltCmd.eOn);
PlantCtrl.AssignAggregate1x(nPltOpMode := E_BA_AC_OpMod01.eCoolDownProtection,			iAgg1Ref := SuAFan, nAgg1OpMode := E_BA_MdltCmd.eOn);
PlantCtrl.AssignAggregate1x(nPltOpMode := E_BA_AC_OpMod01.eOverHeatingProtection,		iAgg1Ref := SuAFan, nAgg1OpMode := E_BA_MdltCmd.eOn);
PlantCtrl.AssignAggregate1x(nPltOpMode := E_BA_AC_OpMod01.eFrost,						iAgg1Ref := SuAFan, nAgg1OpMode := E_BA_MdltCmd.eOff);
PlantCtrl.AssignAggregate1x(nPltOpMode := E_BA_AC_OpMod01.eEmergency,					iAgg1Ref := SuAFan, nAgg1OpMode := E_BA_MdltCmd.eOff);
PlantCtrl.AssignAggregate1x(nPltOpMode := E_BA_AC_OpMod01.eAlarm,						iAgg1Ref := SuAFan, nAgg1OpMode := E_BA_MdltCmd.eOff);
PlantCtrl.AssignAggregate1x(nPltOpMode := E_BA_AC_OpMod01.eForcedVentilation,			iAgg1Ref := SuAFan, nAgg1OpMode := E_BA_MdltCmd.eOn);
PlantCtrl.AssignAggregate1x(nPltOpMode := E_BA_AC_OpMod01.eCentralSwitchOff,			iAgg1Ref := SuAFan, nAgg1OpMode := E_BA_MdltCmd.eOff);
PlantCtrl.AssignAggregate1x(nPltOpMode := E_BA_AC_OpMod01.eSmokeExtractionProgramm,		iAgg1Ref := SuAFan, nAgg1OpMode := E_BA_MdltCmd.eOn);
PlantCtrl.AssignAggregate1x(nPltOpMode := E_BA_AC_OpMod01.eSmokeExtractionSupplyAir,	iAgg1Ref := SuAFan, nAgg1OpMode := E_BA_MdltCmd.eOn);
PlantCtrl.AssignAggregate1x(nPltOpMode := E_BA_AC_OpMod01.eSmokeExtractionExhaustAir,	iAgg1Ref := SuAFan, nAgg1OpMode := E_BA_MdltCmd.eOff);
PlantCtrl.AssignAggregate1x(nPltOpMode := E_BA_AC_OpMod01.eFire,						iAgg1Ref := SuAFan, nAgg1OpMode := E_BA_MdltCmd.eOff);

// Aggregatbetriebsarten in Abhängigkeit von den entsprechenden Anlagenbetriebsarten anwenden:
// Fortluftklappe freigeben in Abhängigkeit von der Anlagenbetriebsart 
// Apply aggregate operation modes dependant on corresponding plant operation modes:
// release exhaust air damper depending on plant operation mode 
PlantCtrl.AssignAggregate1x(nPltOpMode := E_BA_AC_OpMod01.eOff,							iAgg1Ref := ExhADmp, nAgg1OpMode := TO_UDINT(FALSE));
PlantCtrl.AssignAggregate1x(nPltOpMode := E_BA_AC_OpMod01.eOn,							iAgg1Ref := ExhADmp, nAgg1OpMode := TO_UDINT(TRUE));
PlantCtrl.AssignAggregate1x(nPltOpMode := E_BA_AC_OpMod01.eNightCooling,				iAgg1Ref := ExhADmp, nAgg1OpMode := TO_UDINT(TRUE));
PlantCtrl.AssignAggregate1x(nPltOpMode := E_BA_AC_OpMod01.eCoolDownProtection,			iAgg1Ref := ExhADmp, nAgg1OpMode := TO_UDINT(TRUE));
PlantCtrl.AssignAggregate1x(nPltOpMode := E_BA_AC_OpMod01.eOverHeatingProtection,		iAgg1Ref := ExhADmp, nAgg1OpMode := TO_UDINT(TRUE));
PlantCtrl.AssignAggregate1x(nPltOpMode := E_BA_AC_OpMod01.eFrost,						iAgg1Ref := ExhADmp, nAgg1OpMode := TO_UDINT(FALSE));
PlantCtrl.AssignAggregate1x(nPltOpMode := E_BA_AC_OpMod01.eEmergency,					iAgg1Ref := ExhADmp, nAgg1OpMode := TO_UDINT(FALSE));
PlantCtrl.AssignAggregate1x(nPltOpMode := E_BA_AC_OpMod01.eAlarm,						iAgg1Ref := ExhADmp, nAgg1OpMode := TO_UDINT(FALSE));
PlantCtrl.AssignAggregate1x(nPltOpMode := E_BA_AC_OpMod01.eForcedVentilation,			iAgg1Ref := ExhADmp, nAgg1OpMode := TO_UDINT(TRUE));
PlantCtrl.AssignAggregate1x(nPltOpMode := E_BA_AC_OpMod01.eCentralSwitchOff,			iAgg1Ref := ExhADmp, nAgg1OpMode := TO_UDINT(FALSE));
PlantCtrl.AssignAggregate1x(nPltOpMode := E_BA_AC_OpMod01.eSmokeExtractionProgramm,		iAgg1Ref := ExhADmp, nAgg1OpMode := TO_UDINT(TRUE));
PlantCtrl.AssignAggregate1x(nPltOpMode := E_BA_AC_OpMod01.eSmokeExtractionSupplyAir,	iAgg1Ref := ExhADmp, nAgg1OpMode := TO_UDINT(FALSE));
PlantCtrl.AssignAggregate1x(nPltOpMode := E_BA_AC_OpMod01.eSmokeExtractionExhaustAir,	iAgg1Ref := ExhADmp, nAgg1OpMode := TO_UDINT(TRUE));
PlantCtrl.AssignAggregate1x(nPltOpMode := E_BA_AC_OpMod01.eFire,						iAgg1Ref := ExhADmp, nAgg1OpMode := TO_UDINT(FALSE));

// Aggregatbetriebsarten in Abhängigkeit von den entsprechenden Anlagenbetriebsarten anwenden:
// Abluftventilator freigeben in Abhängigkeit von der Anlagenbetriebsart 
// Apply aggregate operation modes dependant on corresponding plant operation modes:
// release extract air fan depending on plant operation mode 
PlantCtrl.AssignAggregate1x(nPltOpMode := E_BA_AC_OpMod01.eOff,							iAgg1Ref := ExtAFan, nAgg1OpMode := E_BA_MdltCmd.eOff);
PlantCtrl.AssignAggregate1x(nPltOpMode := E_BA_AC_OpMod01.eOn,							iAgg1Ref := ExtAFan, nAgg1OpMode := E_BA_MdltCmd.eOn); 
PlantCtrl.AssignAggregate1x(nPltOpMode := E_BA_AC_OpMod01.eNightCooling,				iAgg1Ref := ExtAFan, nAgg1OpMode := E_BA_MdltCmd.eOn); 
PlantCtrl.AssignAggregate1x(nPltOpMode := E_BA_AC_OpMod01.eCoolDownProtection,			iAgg1Ref := ExtAFan, nAgg1OpMode := E_BA_MdltCmd.eOn); 
PlantCtrl.AssignAggregate1x(nPltOpMode := E_BA_AC_OpMod01.eOverHeatingProtection,		iAgg1Ref := ExtAFan, nAgg1OpMode := E_BA_MdltCmd.eOn); 
PlantCtrl.AssignAggregate1x(nPltOpMode := E_BA_AC_OpMod01.eFrost,						iAgg1Ref := ExtAFan, nAgg1OpMode := E_BA_MdltCmd.eOff);
PlantCtrl.AssignAggregate1x(nPltOpMode := E_BA_AC_OpMod01.eEmergency,					iAgg1Ref := ExtAFan, nAgg1OpMode := E_BA_MdltCmd.eOff);
PlantCtrl.AssignAggregate1x(nPltOpMode := E_BA_AC_OpMod01.eAlarm,						iAgg1Ref := ExtAFan, nAgg1OpMode := E_BA_MdltCmd.eOff);
PlantCtrl.AssignAggregate1x(nPltOpMode := E_BA_AC_OpMod01.eForcedVentilation,			iAgg1Ref := ExtAFan, nAgg1OpMode := E_BA_MdltCmd.eOn); 
PlantCtrl.AssignAggregate1x(nPltOpMode := E_BA_AC_OpMod01.eCentralSwitchOff,			iAgg1Ref := ExtAFan, nAgg1OpMode := E_BA_MdltCmd.eOff);
PlantCtrl.AssignAggregate1x(nPltOpMode := E_BA_AC_OpMod01.eSmokeExtractionProgramm,		iAgg1Ref := ExtAFan, nAgg1OpMode := E_BA_MdltCmd.eOn); 
PlantCtrl.AssignAggregate1x(nPltOpMode := E_BA_AC_OpMod01.eSmokeExtractionSupplyAir,	iAgg1Ref := ExtAFan, nAgg1OpMode := E_BA_MdltCmd.eOff);
PlantCtrl.AssignAggregate1x(nPltOpMode := E_BA_AC_OpMod01.eSmokeExtractionExhaustAir,	iAgg1Ref := ExtAFan, nAgg1OpMode := E_BA_MdltCmd.eOn); 
PlantCtrl.AssignAggregate1x(nPltOpMode := E_BA_AC_OpMod01.eFire,						iAgg1Ref := ExtAFan, nAgg1OpMode := E_BA_MdltCmd.eOff);

// Aggregatbetriebsarten in Abhängigkeit von den entsprechenden Anlagenbetriebsarten anwenden:
// Kaskadenregelung freigeben in Abhängigkeit von der Anlagenbetriebsart 
// Apply aggregate operation modes dependant on corresponding plant operation modes:
// release cascade control depending on plant operation mode 
PlantCtrl.AssignAggregate1x(nPltOpMode := E_BA_AC_OpMod01.eOff,							iAgg1Ref := TCasCtrl, nAgg1OpMode := E_BA_MdltCmd.eOff);
PlantCtrl.AssignAggregate1x(nPltOpMode := E_BA_AC_OpMod01.eOn,							iAgg1Ref := TCasCtrl, nAgg1OpMode := E_BA_MdltCmd.eOn);
PlantCtrl.AssignAggregate1x(nPltOpMode := E_BA_AC_OpMod01.eNightCooling,				iAgg1Ref := TCasCtrl, nAgg1OpMode := E_BA_MdltCmd.eOff);
PlantCtrl.AssignAggregate1x(nPltOpMode := E_BA_AC_OpMod01.eCoolDownProtection,			iAgg1Ref := TCasCtrl, nAgg1OpMode := E_BA_MdltCmd.eMax);
PlantCtrl.AssignAggregate1x(nPltOpMode := E_BA_AC_OpMod01.eOverHeatingProtection,		iAgg1Ref := TCasCtrl, nAgg1OpMode := E_BA_MdltCmd.eMin);
PlantCtrl.AssignAggregate1x(nPltOpMode := E_BA_AC_OpMod01.eFrost,						iAgg1Ref := TCasCtrl, nAgg1OpMode := E_BA_MdltCmd.eOff);
PlantCtrl.AssignAggregate1x(nPltOpMode := E_BA_AC_OpMod01.eEmergency,					iAgg1Ref := TCasCtrl, nAgg1OpMode := E_BA_MdltCmd.eOff);
PlantCtrl.AssignAggregate1x(nPltOpMode := E_BA_AC_OpMod01.eAlarm,						iAgg1Ref := TCasCtrl, nAgg1OpMode := E_BA_MdltCmd.eOff);
PlantCtrl.AssignAggregate1x(nPltOpMode := E_BA_AC_OpMod01.eForcedVentilation,			iAgg1Ref := TCasCtrl, nAgg1OpMode := E_BA_MdltCmd.eOn);
PlantCtrl.AssignAggregate1x(nPltOpMode := E_BA_AC_OpMod01.eCentralSwitchOff,			iAgg1Ref := TCasCtrl, nAgg1OpMode := E_BA_MdltCmd.eMin);
PlantCtrl.AssignAggregate1x(nPltOpMode := E_BA_AC_OpMod01.eSmokeExtractionProgramm,		iAgg1Ref := TCasCtrl, nAgg1OpMode := E_BA_MdltCmd.eMin);
PlantCtrl.AssignAggregate1x(nPltOpMode := E_BA_AC_OpMod01.eSmokeExtractionSupplyAir,	iAgg1Ref := TCasCtrl, nAgg1OpMode := E_BA_MdltCmd.eMin);
PlantCtrl.AssignAggregate1x(nPltOpMode := E_BA_AC_OpMod01.eSmokeExtractionExhaustAir,	iAgg1Ref := TCasCtrl, nAgg1OpMode := E_BA_MdltCmd.eOff);
PlantCtrl.AssignAggregate1x(nPltOpMode := E_BA_AC_OpMod01.eFire,						iAgg1Ref := TCasCtrl, nAgg1OpMode := E_BA_MdltCmd.eOff);
END_METHOD

END_FUNCTION_BLOCK

// ---- Templates/POUs/Universal/Control/Hysteresis/FB_BA_Hys_21.TcPOU
{region '#Template'}
	{attribute 'Version' := '1.0.0.0'}
	{attribute 'Tags' := '"LCID": "1031", "Text": "Universal, Control, Hysteresis"'}
	{attribute 'Tags' := '"LCID": "1033", "Text": "Universal, Control, Hysteresis"'}
	{attribute 'Description' := '"LCID": "1031", "Text": "Hysterese"'}
	{attribute 'Description' := '"LCID": "1033", "Text": "Hysteresis"'}
{endregion}
FUNCTION_BLOCK FB_BA_Hys_21 EXTENDS FB_BA_View
VAR_INPUT
	bEn 					: BOOL := TRUE;	
	fIn						: REAL;
END_VAR
VAR_OUTPUT
	bDst					: BOOL;
END_VAR
VAR_INPUT CONSTANT
	HysPreAlarmOn			: FB_BA_AV_Op;		
	HysPreAlarmOff			: FB_BA_AV_Op;		
	HysMainAlarmOn			: FB_BA_AV_Op;		
	HysMainAlarmOff			: FB_BA_AV_Op;	
	DstPreAlarm				: FB_BA_BV;
	DstMainAlarm			: FB_BA_BV;
END_VAR
VAR
	HysPreAlarm				: FB_BA_Swi2P;
	HysMainAlarm			: FB_BA_Swi2P;
END_VAR

SUPER^(); // FB_BA_View
HysPreAlarmOn(); // FB_BA_AV_Op
HysPreAlarmOff(); // FB_BA_AV_Op
HysMainAlarmOn(); // FB_BA_AV_Op
HysMainAlarmOff(); // FB_BA_AV_Op
HysPreAlarm(bEn := bEn, fIn := fIn, fOn := HysPreAlarmOn.fPresentValue, fOff := HysPreAlarmOff.fPresentValue); // FB_BA_Swi2P
DstPreAlarm(bEnPgm := TRUE, bValPgm := HysPreAlarm.bQ); // FB_BA_BV
HysMainAlarm(
    bEn := bEn,
    fIn := fIn,
    fOn := HysMainAlarmOn.fPresentValue,
    fOff := HysMainAlarmOff.fPresentValue); // FB_BA_Swi2P
DstMainAlarm(bEnPgm := TRUE, bValPgm := HysMainAlarm.bQ); // FB_BA_BV
bDst := DstPreAlarm.bEvent OR DstMainAlarm.bEvent;

METHOD FB_init : BOOL
VAR_INPUT
	bInitRetains : BOOL; // if TRUE, the retain variables are initialized (warm start / cold start)
	bInCopyCode : BOOL;  // if TRUE, the instance afterwards gets moved into the copy code (online change)
END_VAR
HysPreAlarmOn.iParent						:= THIS^;
HysPreAlarmOn.iLabel						:= LblUniControl.Hysteresis_PreAlarmLimitMAX;	 
HysPreAlarmOn.sObjectName					:= '{Idx=01}';	
HysPreAlarmOn.eUnit							:= E_BA_Unit.ePressure_Pascals;							 	 
HysPreAlarmOn.fValueRm						:= 200;			
HysPreAlarmOn.fCOVIncrement					:= BA2_Param.fDefCOVIncrement;		

HysPreAlarmOff.iParent						:= THIS^;
HysPreAlarmOff.iLabel						:= LblUniControl.Hysteresis_PreAlarmLimitMIN;	 
HysPreAlarmOff.sObjectName					:= '{Idx=01}';	
HysPreAlarmOff.eUnit						:= E_BA_Unit.ePressure_Pascals;							 	 
HysPreAlarmOff.fValueRm						:= 150;			
HysPreAlarmOff.fCOVIncrement				:= BA2_Param.fDefCOVIncrement;		
							
HysMainAlarmOn.iParent						:= THIS^;
HysMainAlarmOn.iLabel						:= LblUniControl.Hysteresis_MainAlarmLimitMAX; 
HysMainAlarmOn.sObjectName					:= '{Idx=02}';								 	 
HysMainAlarmOn.eUnit						:= E_BA_Unit.ePressure_Pascals;
HysMainAlarmOn.fValueRm						:= 350;			
HysMainAlarmOn.fCOVIncrement				:= BA2_Param.fDefCOVIncrement;		
							
HysMainAlarmOff.iParent						:= THIS^;
HysMainAlarmOff.iLabel						:= LblUniControl.Hysteresis_MainAlarmLimitMIN; 
HysMainAlarmOff.sObjectName					:= '{Idx=02}';								 	 
HysMainAlarmOff.eUnit						:= E_BA_Unit.ePressure_Pascals;
HysMainAlarmOff.fValueRm					:= 300;			
HysMainAlarmOff.fCOVIncrement				:= BA2_Param.fDefCOVIncrement;		

DstPreAlarm.iParent							:= THIS^;
DstPreAlarm.iLabel							:= LblUniControl.Hysteresis_PreAlarmFault;			
DstPreAlarm.sObjectName						:= '{Idx=01}';	
DstPreAlarm.bEnOutOfService					:= FALSE;
DstPreAlarm.sActiveText 					:= txtEvent_Maintenace;
DstPreAlarm.sInactiveText 					:= txtEvent_Normal;
DstPreAlarm.nStateChangeCount				:= 0;
DstPreAlarm.nActiveTimeElapsed				:= 0;
DstPreAlarm.nMinimumOnTime					:= 0;
DstPreAlarm.nMinimumOffTime					:= 0;
DstPreAlarm.bEnManualRm						:= FALSE;	//	Priority  8	
DstPreAlarm.bValManualRm					:= FALSE;	//	Priority  8
DstPreAlarm.bDefaultValue					:= FALSE;
DstPreAlarm.nEventClassID					:= EventClasses.MaintenanceSimple;
DstPreAlarm.stTimeDelay.nToNormal			:= BA2_Param.nDefTimeDelay_ToNormal;
DstPreAlarm.stTimeDelay.nToAbnormal			:= BA2_Param.nDefTimeDelay_ToAbnormal;
DstPreAlarm.bAlarmValue						:= TRUE;
DstPreAlarm.bAcknowledgeRm					:= FALSE;		
DstPreAlarm.aEventTransitionText[1]			:= txtEvent_Disturb;
DstPreAlarm.aEventTransitionText[2]			:= txtEvent_None;
DstPreAlarm.aEventTransitionText[3]			:= txtEvent_Normal;
DstPreAlarm.bEventDetectionEnable			:= TRUE;
DstPreAlarm.eEnPlantLock					:= E_BA_LockPriority.eNoLock;	

DstMainAlarm.iParent						:= THIS^;
DstMainAlarm.iLabel							:= LblUniControl.Hysteresis_MainAlarmFault;			
DstMainAlarm.sObjectName					:= '{Idx=02}';	
DstMainAlarm.bEnOutOfService				:= FALSE;
DstMainAlarm.sActiveText 					:= txtEvent_Triggered;
DstMainAlarm.sInactiveText 					:= txtEvent_Normal;
DstMainAlarm.nStateChangeCount				:= 0;
DstMainAlarm.nActiveTimeElapsed				:= 0;
DstMainAlarm.nMinimumOnTime					:= 0;
DstMainAlarm.nMinimumOffTime				:= 0;
DstMainAlarm.bEnManualRm					:= FALSE;	//	Priority  8	
DstMainAlarm.bValManualRm					:= FALSE;	//	Priority  8
DstMainAlarm.bDefaultValue					:= FALSE;
DstMainAlarm.nEventClassID					:= EventClasses.AlarmTechnicalExtended;
DstMainAlarm.stTimeDelay.nToNormal			:= BA2_Param.nDefTimeDelay_ToNormal;
DstMainAlarm.stTimeDelay.nToAbnormal		:= BA2_Param.nDefTimeDelay_ToAbnormal;
DstMainAlarm.bAlarmValue					:= TRUE;
DstMainAlarm.bAcknowledgeRm					:= FALSE;		
DstMainAlarm.aEventTransitionText[1]		:= txtEvent_Triggered;
DstMainAlarm.aEventTransitionText[2]		:= txtEvent_Error;
DstMainAlarm.aEventTransitionText[3]		:= txtEvent_Normal;
DstMainAlarm.bEventDetectionEnable			:= TRUE;
DstMainAlarm.eEnPlantLock					:= E_BA_LockPriority.eNoLock;
END_METHOD

END_FUNCTION_BLOCK

// ---- Templates/POUs/Trade/AC/General/FB_BA_AC_SumNgtCol.TcPOU
{region '#Template'}
	{attribute 'Version' := '1.0.0.0'}
	{attribute 'Tags' := '"LCID": "1031", "Text": "AC, General, night cooling"'}
	{attribute 'Tags' := '"LCID": "1033", "Text": "AC, General, night cooling"'}
	{attribute 'Description' := '"LCID": "1031", "Text": "Nachtkühlung"'}
	{attribute 'Description' := '"LCID": "1033", "Text": "night cooling"'}
{endregion}
FUNCTION_BLOCK FB_BA_AC_SumNgtCol EXTENDS FB_BA_View
VAR_INPUT
	fTRm					: REAL;
	fSpRm					: REAL;
	fTWth					: REAL;		
END_VAR
VAR_OUTPUT
	bQ						: BOOL;
END_VAR
VAR_INPUT CONSTANT
	WthTLoLmt				: FB_BA_AV_Op;	
	RmTHys					: FB_BA_AV_Op;	
	SwiOnDiffT				: FB_BA_AV_Op;	
	SwiOffDiffT				: FB_BA_AV_Op;	
	Q						: FB_BA_BV_Op;																					
	Sched					: FB_BA_SchedM;
END_VAR
VAR
	NgtColFnct				: FB_BA_NgtCol;
END_VAR

SUPER^(); // FB_BA_View
Sched(); // FB_BA_SchedM
WthTLoLmt(); // FB_BA_AV_Op
RmTHys(); // FB_BA_AV_Op
SwiOnDiffT(); // FB_BA_AV_Op
SwiOffDiffT(); // FB_BA_AV_Op
NgtColFnct(
    bEn := Sched.nPresentValue = E_BA_OnOff.eOn,
    fTOts := fTWth,
    fTRm := fTRm,
    fSpRm := fSpRm,
    fTOtsLoLmt := WthTLoLmt.fPresentValue,
    fTRmHys := RmTHys.fPresentValue,
    fSwiOnDiffT := SwiOnDiffT.fPresentValue,
    fSwiOffDiffT := SwiOffDiffT.fPresentValue); // FB_BA_NgtCol
Q(bValuePgm := NgtColFnct.bQ); // FB_BA_BV_Op
bQ := Q.bPresentValue;

METHOD FB_init : BOOL
VAR_INPUT
	bInitRetains : BOOL; // if TRUE, the retain variables are initialized (warm start / cold start)
	bInCopyCode : BOOL;  // if TRUE, the instance afterwards gets moved into the copy code (online change)
END_VAR
WthTLoLmt.iParent			:= THIS^;
WthTLoLmt.iLabel			:= LblCmpAC.General_SumNgtCol_WthTLoLmt;			
WthTLoLmt.sObjectName		:= '{Idx=01}';								 	 
WthTLoLmt.eUnit				:= E_BA_Unit.eTemperature_DegreesCelsius;  
WthTLoLmt.fValueRm			:= 9.0;

RmTHys.iParent				:= THIS^;
RmTHys.iLabel				:= LblCmpAC.General_SumNgtCol_RmTHys;			
RmTHys.sObjectName			:= '{Idx=01}';								 	 
RmTHys.eUnit				:= E_BA_Unit.eTemperature_DegreesCelsius;  
RmTHys.fValueRm				:= 2.0;

SwiOnDiffT.iParent			:= THIS^;
SwiOnDiffT.iLabel			:= LblCmpAC.General_SumNgtCol_SwiOnDiffT;			
SwiOnDiffT.sObjectName		:= '{Idx=01}';								 	 
SwiOnDiffT.eUnit			:= E_BA_Unit.eTemperature_DegreesCelsius;  
SwiOnDiffT.fValueRm			:= 7.0;

SwiOffDiffT.iParent			:= THIS^;
SwiOffDiffT.iLabel			:= LblCmpAC.General_SumNgtCol_SwiOffDiffT;			
SwiOffDiffT.sObjectName		:= '{Idx=02}';								 	 
SwiOffDiffT.eUnit			:= E_BA_Unit.eTemperature_DegreesCelsius;  
SwiOffDiffT.fValueRm		:= 5.0;

Q.iParent					:= THIS^;
Q.iLabel					:= LblCmpAC.General_SumNgtCol_Q;												 
Q.sObjectName				:= '{Idx=01}';
Q.sInactiveText				:= txtEvent_Off;
Q.sActiveText				:= txtEvent_On;
Q.bValueRm					:= FALSE;								
Q.eToggleMode 				:= E_BA_ToggleMode.eSwitch;

Sched.iParent											:= THIS^;
Sched.iLabel											:= LblCmpAC.General_SumNgtCol_Sched;							
Sched.sObjectName										:= '{Idx=01}';		
Sched.aStateText[1]										:= txtEvent_Off;
Sched.aStateText[2]										:= txtEvent_On;
Sched.nPredictTime										:= 0;
Sched.nDefaultValue										:= E_BA_OnOff.eOff;
Sched.bWriteWeekly										:= FALSE;
//	Monday
Sched.aWeek[E_BA_Weekday.eMonday,1].eState				:= E_BA_SchedEntryState.eValue;
Sched.aWeek[E_BA_Weekday.eMonday,1].uValue.udiVal		:= E_BA_OnOff.eOn;
Sched.aWeek[E_BA_Weekday.eMonday,1].stTime.nHour		:= 1;
Sched.aWeek[E_BA_Weekday.eMonday,1].stTime.nMinute		:= 0;
Sched.aWeek[E_BA_Weekday.eMonday,1].stTime.nSecond		:= 0;
Sched.aWeek[E_BA_Weekday.eMonday,2].eState				:= E_BA_SchedEntryState.eValue;
Sched.aWeek[E_BA_Weekday.eMonday,2].uValue.udiVal		:= E_BA_OnOff.eOff;
Sched.aWeek[E_BA_Weekday.eMonday,2].stTime.nHour		:= 5;
Sched.aWeek[E_BA_Weekday.eMonday,2].stTime.nMinute		:= 0;
Sched.aWeek[E_BA_Weekday.eMonday,2].stTime.nSecond		:= 0;
Sched.aWeek[E_BA_Weekday.eMonday,3].eState				:= E_BA_SchedEntryState.eValue;
Sched.aWeek[E_BA_Weekday.eMonday,3].uValue.udiVal		:= E_BA_OnOff.eOff;
Sched.aWeek[E_BA_Weekday.eMonday,3].stTime.nHour		:= 0;
Sched.aWeek[E_BA_Weekday.eMonday,3].stTime.nMinute		:= 0;
Sched.aWeek[E_BA_Weekday.eMonday,3].stTime.nSecond		:= 0;
//	Tuesday
Sched.aWeek[E_BA_Weekday.eTuesday,1].eState				:= E_BA_SchedEntryState.eValue;
Sched.aWeek[E_BA_Weekday.eTuesday,1].uValue.udiVal		:= E_BA_OnOff.eOn;
Sched.aWeek[E_BA_Weekday.eTuesday,1].stTime.nHour		:= 1;
Sched.aWeek[E_BA_Weekday.eTuesday,1].stTime.nMinute		:= 0;
Sched.aWeek[E_BA_Weekday.eTuesday,1].stTime.nSecond		:= 0;
Sched.aWeek[E_BA_Weekday.eTuesday,2].eState				:= E_BA_SchedEntryState.eValue;
Sched.aWeek[E_BA_Weekday.eTuesday,2].uValue.udiVal		:= E_BA_OnOff.eOff;
Sched.aWeek[E_BA_Weekday.eTuesday,2].stTime.nHour		:= 5;
Sched.aWeek[E_BA_Weekday.eTuesday,2].stTime.nMinute		:= 0;
Sched.aWeek[E_BA_Weekday.eTuesday,2].stTime.nSecond		:= 0;
Sched.aWeek[E_BA_Weekday.eTuesday,3].eState				:= E_BA_SchedEntryState.eValue;
Sched.aWeek[E_BA_Weekday.eTuesday,3].uValue.udiVal		:= E_BA_OnOff.eOff;
Sched.aWeek[E_BA_Weekday.eTuesday,3].stTime.nHour		:= 0;
Sched.aWeek[E_BA_Weekday.eTuesday,3].stTime.nMinute		:= 0;
Sched.aWeek[E_BA_Weekday.eTuesday,3].stTime.nSecond		:= 0;
//	Wednesday
Sched.aWeek[E_BA_Weekday.eWednesday,1].eState			:= E_BA_SchedEntryState.eValue;
Sched.aWeek[E_BA_Weekday.eWednesday,1].uValue.udiVal	:= E_BA_OnOff.eOn;
Sched.aWeek[E_BA_Weekday.eWednesday,1].stTime.nHour		:= 1;
Sched.aWeek[E_BA_Weekday.eWednesday,1].stTime.nMinute	:= 0;
Sched.aWeek[E_BA_Weekday.eWednesday,1].stTime.nSecond	:= 0;
Sched.aWeek[E_BA_Weekday.eWednesday,2].eState			:= E_BA_SchedEntryState.eValue;
Sched.aWeek[E_BA_Weekday.eWednesday,2].uValue.udiVal	:= E_BA_OnOff.eOff;
Sched.aWeek[E_BA_Weekday.eWednesday,2].stTime.nHour		:= 5;
Sched.aWeek[E_BA_Weekday.eWednesday,2].stTime.nMinute	:= 0;
Sched.aWeek[E_BA_Weekday.eWednesday,2].stTime.nSecond	:= 0;
Sched.aWeek[E_BA_Weekday.eWednesday,3].eState			:= E_BA_SchedEntryState.eValue;
Sched.aWeek[E_BA_Weekday.eWednesday,3].uValue.udiVal	:= E_BA_OnOff.eOff;
Sched.aWeek[E_BA_Weekday.eWednesday,3].stTime.nHour		:= 0;
Sched.aWeek[E_BA_Weekday.eWednesday,3].stTime.nMinute	:= 0;
Sched.aWeek[E_BA_Weekday.eWednesday,3].stTime.nSecond	:= 0;
//	Thursday
Sched.aWeek[E_BA_Weekday.eThursday,1].eState			:= E_BA_SchedEntryState.eValue;
Sched.aWeek[E_BA_Weekday.eThursday,1].uValue.udiVal		:= E_BA_OnOff.eOn;
Sched.aWeek[E_BA_Weekday.eThursday,1].stTime.nHour		:= 1;
Sched.aWeek[E_BA_Weekday.eThursday,1].stTime.nMinute	:= 0;
Sched.aWeek[E_BA_Weekday.eThursday,1].stTime.nSecond	:= 0;
Sched.aWeek[E_BA_Weekday.eThursday,2].eState			:= E_BA_SchedEntryState.eValue;
Sched.aWeek[E_BA_Weekday.eThursday,2].uValue.udiVal		:= E_BA_OnOff.eOff;
Sched.aWeek[E_BA_Weekday.eThursday,2].stTime.nHour		:= 5;
Sched.aWeek[E_BA_Weekday.eThursday,2].stTime.nMinute	:= 0;
Sched.aWeek[E_BA_Weekday.eThursday,2].stTime.nSecond	:= 0;
Sched.aWeek[E_BA_Weekday.eThursday,3].eState			:= E_BA_SchedEntryState.eValue;
Sched.aWeek[E_BA_Weekday.eThursday,3].uValue.udiVal		:= E_BA_OnOff.eOff;
Sched.aWeek[E_BA_Weekday.eThursday,3].stTime.nHour		:= 0;
Sched.aWeek[E_BA_Weekday.eThursday,3].stTime.nMinute	:= 0;
Sched.aWeek[E_BA_Weekday.eThursday,3].stTime.nSecond	:= 0;
//	Friday
Sched.aWeek[E_BA_Weekday.eFriday,1].eState				:= E_BA_SchedEntryState.eValue;
Sched.aWeek[E_BA_Weekday.eFriday,1].uValue.udiVal		:= E_BA_OnOff.eOn;
Sched.aWeek[E_BA_Weekday.eFriday,1].stTime.nHour		:= 1;
Sched.aWeek[E_BA_Weekday.eFriday,1].stTime.nMinute		:= 0;
Sched.aWeek[E_BA_Weekday.eFriday,1].stTime.nSecond		:= 0;
Sched.aWeek[E_BA_Weekday.eFriday,2].eState				:= E_BA_SchedEntryState.eValue;
Sched.aWeek[E_BA_Weekday.eFriday,2].uValue.udiVal		:= E_BA_OnOff.eOff;
Sched.aWeek[E_BA_Weekday.eFriday,2].stTime.nHour		:= 5;
Sched.aWeek[E_BA_Weekday.eFriday,2].stTime.nMinute		:= 0;
Sched.aWeek[E_BA_Weekday.eFriday,2].stTime.nSecond		:= 0;
Sched.aWeek[E_BA_Weekday.eFriday,3].eState				:= E_BA_SchedEntryState.eValue;
Sched.aWeek[E_BA_Weekday.eFriday,3].uValue.udiVal		:= E_BA_OnOff.eOff;
Sched.aWeek[E_BA_Weekday.eFriday,3].stTime.nHour		:= 0;
Sched.aWeek[E_BA_Weekday.eFriday,3].stTime.nMinute		:= 0;
Sched.aWeek[E_BA_Weekday.eFriday,3].stTime.nSecond		:= 0;
Sched.bWriteException									:= FALSE;
END_METHOD

END_FUNCTION_BLOCK

// ---- Templates/POUs/Trade/AC/General/FB_BA_AC_OpMod1St.TcPOU
{region '#Template'}
	{attribute 'Version' := '1.0.0.0'}
	{attribute 'Tags' := '"LCID": "1031", "Text": "AC, General, AHU, Operating mode"'}
	{attribute 'Tags' := '"LCID": "1033", "Text": "AC, General, AHU, Operating mode"'}
	{attribute 'Description' := '"LCID": "1031", "Text": "Betriebsart"'}
	{attribute 'Description' := '"LCID": "1033", "Text": "Operating mode"'}
{endregion}
FUNCTION_BLOCK FB_BA_AC_OpMod1St EXTENDS FB_BA_View
VAR_INPUT
	bSmExttSuA				: BOOL;	// smoke extraction supply air
	bSmExttExhA				: BOOL;	// smoke extraction exhaust air
	bFireDetc				: BOOL;	// fire detection alarm
	bForcVent				: BOOL;	// Forced ventilation
	bEmgOff					: BOOL;	// emergency stop
	bFrst					: BOOL;	// Frost protection is active
	bCentSwiOff				: BOOL;	// Central switch-off	
	bAlmShutOff				: BOOL;	// Shut Off plant collective alarm
	bNgtCol					: BOOL;	// Summer night cooling
	bColDwnPrtc				: BOOL;	// Cooling down protection
	bOvrHtgPrtc				: BOOL;	// Overheating protection
END_VAR
VAR_OUTPUT
	eOpMode					: E_BA_AC_OpMod01;
END_VAR
VAR_INPUT CONSTANT
	OpModMan				: FB_BA_MV_Op;	
	Sched					: FB_BA_SchedM;
	OpModPr					: FB_BA_MV_Op;
END_VAR
VAR
	PrioSwi					: FB_BA_PrioSwi_UDI24;
END_VAR

